LIN {X 0,Y 186.458,Z 664.253,A -85,B 0,C 180,E1 -22354.51,E2 -22354.51} C_VEL
LIN {X 0,Y 188.519,Z 666.422,A -85,B 0,C 180,E1 -22355.462,E2 -22355.462} C_VEL
LIN {X 0,Y 189.961,Z 668.387,A -85,B 0,C 180,E1 -22356.131,E2 -22356.131} C_VEL
LIN {X 0,Y 193.772,Z 674.141,A -85,B 0,C 180,E1 -22357.839,E2 -22357.839} C_VEL
LIN {X 0,Y 198,Z 681.171,A -85,B 0,C 180,E1 -22359.627,E2 -22359.627} C_VEL
LIN {X 0,Y 202.989,Z 690.013,A -85,B 0,C 180,E1 -22361.599,E2 -22361.599} C_VEL
LIN {X 0,Y 209.393,Z 702.579,A -85,B 0,C 180,E1 -22363.96,E2 -22363.96} C_VEL
LIN {X 0,Y 214.813,Z 715.083,A -85,B 0,C 180,E1 -22365.866,E2 -22365.866} C_VEL
LIN {X 0,Y 219.093,Z 726.699,A -85,B 0,C 180,E1 -22367.342,E2 -22367.342} C_VEL
LIN {X 0,Y 219.562,Z 732.346,A -85,B 0,C 180,E1 -22367.681,E2 -22367.681} C_VEL
LIN {X 0,Y 219.234,Z 736.244,A -85,B 0,C 180,E1 -22367.773,E2 -22367.773} C_VEL
LIN {X 0,Y 217.38,Z 743.918,A -85,B 0,C 180,E1 -22367.69,E2 -22367.69} C_VEL
LIN {X 0,Y 213.263,Z 757.174,A -85,B 0,C 180,E1 -22367.338,E2 -22367.338} C_VEL
LIN {X 0,Y 212.359,Z 763.033,A -85,B 0,C 180,E1 -22367.387,E2 -22367.387} C_VEL
LIN {X 0,Y 210.033,Z 802.061,A -85,B 0,C 180,E1 -22368.634,E2 -22368.634} C_VEL
LIN {X 0,Y 208.26,Z 816.506,A -85,B 0,C 180,E1 -22369.407,E2 -22369.407} C_VEL
LIN {X 0,Y 205.986,Z 829.249,A -85,B 0,C 180,E1 -22370.387,E2 -22370.387} C_VEL
LIN {X 0,Y 203.017,Z 842.443,A -85,B 0,C 180,E1 -22371.772,E2 -22371.772} C_VEL
LIN {X 0,Y 199.554,Z 855.196,A -85,B 0,C 180,E1 -22373.536,E2 -22373.536} C_VEL
LIN {X 0,Y 196.163,Z 866.216,A -85,B 0,C 180,E1 -22375.49,E2 -22375.49} C_VEL
LIN {X 0,Y 192.35,Z 877.477,A -85,B 0,C 180,E1 -22378.008,E2 -22378.008} C_VEL
LIN {X 0,Y 188.32,Z 888.046,A -85,B 0,C 180,E1 -22380.977,E2 -22380.977} C_VEL
LIN {X 0,Y 184.98,Z 896.778,A -85,B 0,C 180,E1 -22384.092,E2 -22384.092} C_VEL
LIN {X 0,Y 182.131,Z 904.027,A -85,B 0,C 180,E1 -22387.302,E2 -22387.302} C_VEL
LIN {X 0,Y 179.919,Z 910.061,A -85,B 0,C 180,E1 -22390.608,E2 -22390.608} C_VEL
LIN {X 0,Y 178.213,Z 915.047,A -85,B 0,C 180,E1 -22393.975,E2 -22393.975} C_VEL
LIN {X 0,Y 176.719,Z 920.187,A -85,B 0,C 180,E1 -22398.53,E2 -22398.53} C_VEL
LIN {X 0,Y 176.133,Z 923.805,A -85,B 0,C 180,E1 -22403.125,E2 -22403.125} C_VEL
LIN {X 0,Y 176.096,Z 925.996,A -85,B 0,C 180,E1 -22407.712,E2 -22407.712} C_VEL
LIN {X 0,Y 176.209,Z 926.574,A -85,B 0,C 180,E1 -22410,E2 -22410} C_VEL
LIN {X 0,Y 176.02,Z 926.688,A -85,B 0,C 180,E1 -22414.58,E2 -22414.58} C_VEL
LIN {X 0,Y 176.329,Z 925.467,A -85,B 0,C 180,E1 -22419.174,E2 -22419.174} C_VEL
LIN {X 0,Y 177.401,Z 922.904,A -85,B 0,C 180,E1 -22423.751,E2 -22423.751} C_VEL
LIN {X 0,Y 179.558,Z 918.924,A -85,B 0,C 180,E1 -22428.247,E2 -22428.247} C_VEL
LIN {X 0,Y 182.331,Z 913.868,A -85,B 0,C 180,E1 -22432.32,E2 -22432.32} C_VEL
LIN {X 0,Y 186.083,Z 907.172,A -85,B 0,C 180,E1 -22436.345,E2 -22436.345} C_VEL
LIN {X 0,Y 190.386,Z 899.447,A -85,B 0,C 180,E1 -22439.89,E2 -22439.89} C_VEL
LIN {X 0,Y 194.724,Z 891.411,A -85,B 0,C 180,E1 -22442.778,E2 -22442.778} C_VEL
LIN {X 0,Y 199.516,Z 881.745,A -85,B 0,C 180,E1 -22445.536,E2 -22445.536} C_VEL
LIN {X 0,Y 204.224,Z 871.045,A -85,B 0,C 180,E1 -22447.961,E2 -22447.961} C_VEL
LIN {X 0,Y 208.917,Z 859.221,A -85,B 0,C 180,E1 -22450.043,E2 -22450.043} C_VEL
LIN {X 0,Y 213.409,Z 846.062,A -85,B 0,C 180,E1 -22451.826,E2 -22451.826} C_VEL
LIN {X 0,Y 217.08,Z 833.039,A -85,B 0,C 180,E1 -22453.151,E2 -22453.151} C_VEL
LIN {X 0,Y 220.206,Z 818.846,A -85,B 0,C 180,E1 -22454.199,E2 -22454.199} C_VEL
LIN {X 0,Y 222.422,Z 804.381,A -85,B 0,C 180,E1 -22454.941,E2 -22454.941} C_VEL
LIN {X 0,Y 224.005,Z 785.386,A -85,B 0,C 180,E1 -22455.543,E2 -22455.543} C_VEL
LIN {X 0,Y 226.866,Z 740.906,A -85,B 0,C 180,E1 -22456.815,E2 -22456.815} C_VEL
LIN {X 0,Y 223.203,Z 731.743,A -85,B 0,C 180,E1 -22458.353,E2 -22458.353} C_VEL
LIN {X 0,Y 218.442,Z 721.156,A -85,B 0,C 180,E1 -22460.444,E2 -22460.444} C_VEL
LIN {X 0,Y 212.911,Z 710.324,A -85,B 0,C 180,E1 -22463.05,E2 -22463.05} C_VEL
LIN {X 0,Y 207.489,Z 700.825,A -85,B 0,C 180,E1 -22465.86,E2 -22465.86} C_VEL
LIN {X 0,Y 204.073,Z 695.198,A -85,B 0,C 180,E1 -22467.81,E2 -22467.81} C_VEL
LIN {X 0,Y 201.093,Z 690.54,A -85,B 0,C 180,E1 -22469.652,E2 -22469.652} C_VEL
LIN {X 0,Y 197.75,Z 685.547,A -85,B 0,C 180,E1 -22471.914,E2 -22471.914} C_VEL
LIN {X 0,Y 193.988,Z 680.428,A -85,B 0,C 180,E1 -22474.764,E2 -22474.764} C_VEL
LIN {X 0,Y 193.438,Z 679.67,A -85,B 0,C 180,E1 -22475.22,E2 -22475.22} C_VEL
LIN {X 0,Y 190.753,Z 677.183,A -85,B 0,C 180,E1 -22477.501,E2 -22477.501} C_VEL
LIN {X 0,Y 189.274,Z 674.416,A -85,B 0,C 180,E1 -22479.061,E2 -22479.061} C_VEL
LIN {X 0,Y 186.17,Z 672.169,A -85,B 0,C 180,E1 -22482.423,E2 -22482.423} C_VEL
LIN {X 0,Y 184.562,Z 669.313,A -85,B 0,C 180,E1 -22484.824,E2 -22484.824} C_VEL
LIN {X 0,Y 184.282,Z 668.398,A -85,B 0,C 180,E1 -22485.366,E2 -22485.366} C_VEL
LIN {X 0,Y 180.317,Z 665.407,A -85,B 0,C 180,E1 -22497.767,E2 -22497.767} C_VEL
LIN {X 0,Y 180.526,Z 665.448,A -85,B 0,C 180,E1 -22500.558,E2 -22500.558} C_VEL
LIN {X 0,Y 182.784,Z 667.786,A -85,B 0,C 180,E1 -22507.735,E2 -22507.735} C_VEL
LIN {X 0,Y 184.46,Z 668.55,A -85,B 0,C 180,E1 -22510.486,E2 -22510.486} C_VEL
LIN {X 0,Y 185.451,Z 671.116,A -85,B 0,C 180,E1 -22512.17,E2 -22512.17} C_VEL
LIN {X 0,Y 187.688,Z 673.465,A -85,B 0,C 180,E1 -22514.919,E2 -22514.919} C_VEL
LIN {X 0,Y 189.332,Z 674.523,A -85,B 0,C 180,E1 -22516.581,E2 -22516.581} C_VEL
LIN {X 0,Y 191.05,Z 677.607,A -85,B 0,C 180,E1 -22518.36,E2 -22518.36} C_VEL
LIN {X 0,Y 193.858,Z 680.189,A -85,B 0,C 180,E1 -22520.7,E2 -22520.7} C_VEL
LIN {X 0,Y 196.314,Z 683.711,A -85,B 0,C 180,E1 -22522.635,E2 -22522.635} C_VEL
LIN {X 0,Y 198.092,Z 685.527,A -85,B 0,C 180,E1 -22523.864,E2 -22523.864} C_VEL
LIN {X 0,Y 200.895,Z 689.24,A -85,B 0,C 180,E1 -22525.723,E2 -22525.723} C_VEL
LIN {X 0,Y 205.468,Z 695.423,A -85,B 0,C 180,E1 -22528.447,E2 -22528.447} C_VEL
LIN {X 0,Y 210.739,Z 702.824,A -85,B 0,C 180,E1 -22531.222,E2 -22531.222} C_VEL
LIN {X 0,Y 217.232,Z 712.976,A -85,B 0,C 180,E1 -22534.274,E2 -22534.274} C_VEL
LIN {X 0,Y 223.438,Z 723.698,A -85,B 0,C 180,E1 -22536.899,E2 -22536.899} C_VEL
LIN {X 0,Y 227.451,Z 731.558,A -85,B 0,C 180,E1 -22538.491,E2 -22538.491} C_VEL
LIN {X 0,Y 223.562,Z 789.522,A -85,B 0,C 180,E1 -22540.18,E2 -22540.18} C_VEL
LIN {X 0,Y 221.655,Z 803.905,A -85,B 0,C 180,E1 -22540.886,E2 -22540.886} C_VEL
LIN {X 0,Y 218.999,Z 817.921,A -85,B 0,C 180,E1 -22541.916,E2 -22541.916} C_VEL
LIN {X 0,Y 215.767,Z 830.231,A -85,B 0,C 180,E1 -22543.083,E2 -22543.083} C_VEL
LIN {X 0,Y 211.746,Z 843.508,A -85,B 0,C 180,E1 -22544.81,E2 -22544.81} C_VEL
LIN {X 0,Y 207.507,Z 854.961,A -85,B 0,C 180,E1 -22546.698,E2 -22546.698} C_VEL
LIN {X 0,Y 203.105,Z 865.457,A -85,B 0,C 180,E1 -22548.894,E2 -22548.894} C_VEL
LIN {X 0,Y 198.737,Z 874.93,A -85,B 0,C 180,E1 -22551.396,E2 -22551.396} C_VEL
LIN {X 0,Y 193.842,Z 884.419,A -85,B 0,C 180,E1 -22554.543,E2 -22554.543} C_VEL
LIN {X 0,Y 189.238,Z 892.563,A -85,B 0,C 180,E1 -22558.047,E2 -22558.047} C_VEL
LIN {X 0,Y 185.363,Z 899.091,A -85,B 0,C 180,E1 -22561.71,E2 -22561.71} C_VEL
LIN {X 0,Y 181.765,Z 904.858,A -85,B 0,C 180,E1 -22566.047,E2 -22566.047} C_VEL
LIN {X 0,Y 179.351,Z 908.731,A -85,B 0,C 180,E1 -22570.131,E2 -22570.131} C_VEL
LIN {X 0,Y 177.673,Z 911.216,A -85,B 0,C 180,E1 -22573.926,E2 -22573.926} C_VEL
LIN {X 0,Y 176.494,Z 912.899,A -85,B 0,C 180,E1 -22578.516,E2 -22578.516} C_VEL
LIN {X 0,Y 176.125,Z 913.253,A -85,B 0,C 180,E1 -22583.125,E2 -22583.125} C_VEL
LIN {X 0,Y 176.143,Z 912.827,A -85,B 0,C 180,E1 -22585.948,E2 -22585.948} C_VEL
LIN {X 0,Y 176.326,Z 911.339,A -85,B 0,C 180,E1 -22590,E2 -22590} C_VEL
LIN {X 0,Y 177.015,Z 908.405,A -85,B 0,C 180,E1 -22594.555,E2 -22594.555} C_VEL
LIN {X 0,Y 178.587,Z 904.042,A -85,B 0,C 180,E1 -22599.057,E2 -22599.057} C_VEL
LIN {X 0,Y 180.536,Z 898.946,A -85,B 0,C 180,E1 -22602.919,E2 -22602.919} C_VEL
LIN {X 0,Y 183.049,Z 892.471,A -85,B 0,C 180,E1 -22606.736,E2 -22606.736} C_VEL
LIN {X 0,Y 186.249,Z 884.467,A -85,B 0,C 180,E1 -22610.429,E2 -22610.429} C_VEL
LIN {X 0,Y 189.769,Z 876.064,A -85,B 0,C 180,E1 -22613.461,E2 -22613.461} C_VEL
LIN {X 0,Y 193.576,Z 865.93,A -85,B 0,C 180,E1 -22616.408,E2 -22616.408} C_VEL
LIN {X 0,Y 197.334,Z 854.598,A -85,B 0,C 180,E1 -22619.029,E2 -22619.029} C_VEL
LIN {X 0,Y 200.212,Z 844.74,A -85,B 0,C 180,E1 -22620.889,E2 -22620.889} C_VEL
LIN {X 0,Y 203.414,Z 832.733,A -85,B 0,C 180,E1 -22622.674,E2 -22622.674} C_VEL
LIN {X 0,Y 206.431,Z 819.424,A -85,B 0,C 180,E1 -22624.177,E2 -22624.177} C_VEL
LIN {X 0,Y 208.689,Z 805.589,A -85,B 0,C 180,E1 -22625.368,E2 -22625.368} C_VEL
LIN {X 0,Y 210.399,Z 791.062,A -85,B 0,C 180,E1 -22626.216,E2 -22626.216} C_VEL
LIN {X 0,Y 211.902,Z 767.428,A -85,B 0,C 180,E1 -22627.019,E2 -22627.019} C_VEL
LIN {X 0,Y 214.604,Z 720.39,A -85,B 0,C 180,E1 -22628.444,E2 -22628.444} C_VEL
LIN {X 0,Y 209.401,Z 709.666,A -85,B 0,C 180,E1 -22630.204,E2 -22630.204} C_VEL
LIN {X 0,Y 203.348,Z 698.745,A -85,B 0,C 180,E1 -22632.36,E2 -22632.36} C_VEL
LIN {X 0,Y 197.061,Z 688.675,A -85,B 0,C 180,E1 -22634.769,E2 -22634.769} C_VEL
LIN {X 0,Y 191.638,Z 680.859,A -85,B 0,C 180,E1 -22637.025,E2 -22637.025} C_VEL
LIN {X 0,Y 188.675,Z 676.773,A -85,B 0,C 180,E1 -22638.35,E2 -22638.35} C_VEL
LIN {X 0,Y 186.132,Z 673.147,A -85,B 0,C 180,E1 -22639.561,E2 -22639.561} C_VEL
LIN {X 0,Y 183.199,Z 669.724,A -85,B 0,C 180,E1 -22640.994,E2 -22640.994} C_VEL
LIN {X 0,Y 181.985,Z 667.637,A -85,B 0,C 180,E1 -22641.66,E2 -22641.66} C_VEL
LIN {X 0,Y 179.787,Z 665.649,A -85,B 0,C 180,E1 -22642.793,E2 -22642.793} C_VEL
LIN {X 0,Y 178.655,Z 663.464,A -85,B 0,C 180,E1 -22643.483,E2 -22643.483} C_VEL
LIN {X 0,Y 178.43,Z 662.343,A -85,B 0,C 180,E1 -22643.733,E2 -22643.733} C_VEL
LIN {X 0,Y 178.486,Z 662.376,A -85,B 0,C 180,E1 -22646.546,E2 -22646.546} C_VEL
LIN {X 0,Y 178.447,Z 662.375,A -85,B 0,C 180,E1 -22651.795,E2 -22651.795} C_VEL
LIN {X 0,Y 178.518,Z 662.354,A -85,B 0,C 180,E1 -22654.888,E2 -22654.888} C_VEL
LIN {X 0,Y 178.593,Z 662.347,A -85,B 0,C 180,E1 -22660.814,E2 -22660.814} C_VEL
LIN {X 0,Y 178.647,Z 662.356,A -85,B 0,C 180,E1 -22666.346,E2 -22666.346} C_VEL
LIN {X 0,Y 178.909,Z 662.303,A -85,B 0,C 180,E1 -22670.959,E2 -22670.959} C_VEL
LIN {X 0,Y 179.149,Z 662.292,A -85,B 0,C 180,E1 -22677.751,E2 -22677.751} C_VEL
LIN {X 0,Y 179.369,Z 662.257,A -85,B 0,C 180,E1 -22679.999,E2 -22679.999} C_VEL
LIN {X 0,Y 178.869,Z 662.325,A -85,B 0,C 180,E1 -22684.506,E2 -22684.506} C_VEL
LIN {X 0,Y 178.914,Z 662.322,A -85,B 0,C 180,E1 -22689.04,E2 -22689.04} C_VEL
LIN {X 0,Y 178.66,Z 662.352,A -85,B 0,C 180,E1 -22693.651,E2 -22693.651} C_VEL
LIN {X 0,Y 178.623,Z 662.348,A -85,B 0,C 180,E1 -22699.214,E2 -22699.214} C_VEL
LIN {X 0,Y 178.521,Z 662.367,A -85,B 0,C 180,E1 -22705.114,E2 -22705.114} C_VEL
LIN {X 0,Y 178.524,Z 662.367,A -85,B 0,C 180,E1 -22709.993,E2 -22709.993} C_VEL
LIN {X 0,Y 178.506,Z 662.463,A -85,B 0,C 180,E1 -22710.867,E2 -22710.867} C_VEL
LIN {X 0,Y 179.341,Z 664.986,A -85,B 0,C 180,E1 -22711.445,E2 -22711.445} C_VEL
LIN {X 0,Y 181.355,Z 667.237,A -85,B 0,C 180,E1 -22712.526,E2 -22712.526} C_VEL
LIN {X 0,Y 182.452,Z 668.141,A -85,B 0,C 180,E1 -22713.072,E2 -22713.072} C_VEL
LIN {X 0,Y 184.519,Z 671.443,A -85,B 0,C 180,E1 -22714.168,E2 -22714.168} C_VEL
LIN {X 0,Y 186.456,Z 673.52,A -85,B 0,C 180,E1 -22715.086,E2 -22715.086} C_VEL
LIN {X 0,Y 190.366,Z 679.679,A -85,B 0,C 180,E1 -22716.943,E2 -22716.943} C_VEL
LIN {X 0,Y 195.551,Z 688.346,A -85,B 0,C 180,E1 -22719.219,E2 -22719.219} C_VEL
LIN {X 0,Y 202.299,Z 701.307,A -85,B 0,C 180,E1 -22721.96,E2 -22721.96} C_VEL
LIN {X 0,Y 207.489,Z 712.568,A -85,B 0,C 180,E1 -22723.928,E2 -22723.928} C_VEL
LIN {X 0,Y 212.727,Z 726.005,A -85,B 0,C 180,E1 -22725.851,E2 -22725.851} C_VEL
LIN {X 0,Y 213.798,Z 728.909,A -85,B 0,C 180,E1 -22726.233,E2 -22726.233} C_VEL
LIN {X 0,Y 214.071,Z 733.929,A -85,B 0,C 180,E1 -22726.516,E2 -22726.516} C_VEL
LIN {X 0,Y 212.359,Z 763.033,A -85,B 0,C 180,E1 -22727.387,E2 -22727.387} C_VEL
LIN {X 0,Y 211.505,Z 768.882,A -85,B 0,C 180,E1 -22727.446,E2 -22727.446} C_VEL
LIN {X 0,Y 206.057,Z 787.91,A -85,B 0,C 180,E1 -22727.022,E2 -22727.022} C_VEL
LIN {X 0,Y 205.193,Z 793.759,A -85,B 0,C 180,E1 -22727.081,E2 -22727.081} C_VEL
LIN {X 0,Y 203.858,Z 808.138,A -85,B 0,C 180,E1 -22727.674,E2 -22727.674} C_VEL
LIN {X 0,Y 201.992,Z 820.575,A -85,B 0,C 180,E1 -22728.451,E2 -22728.451} C_VEL
LIN {X 0,Y 199.378,Z 833.862,A -85,B 0,C 180,E1 -22729.63,E2 -22729.63} C_VEL
LIN {X 0,Y 196.088,Z 846.803,A -85,B 0,C 180,E1 -22731.154,E2 -22731.154} C_VEL
LIN {X 0,Y 192.546,Z 858.647,A -85,B 0,C 180,E1 -22732.968,E2 -22732.968} C_VEL
LIN {X 0,Y 188.817,Z 870.156,A -85,B 0,C 180,E1 -22735.25,E2 -22735.25} C_VEL
LIN {X 0,Y 185.62,Z 878.854,A -85,B 0,C 180,E1 -22737.348,E2 -22737.348} C_VEL
LIN {X 0,Y 181.46,Z 889.094,A -85,B 0,C 180,E1 -22740.408,E2 -22740.408} C_VEL
LIN {X 0,Y 178.042,Z 897.603,A -85,B 0,C 180,E1 -22743.635,E2 -22743.635} C_VEL
LIN {X 0,Y 174.615,Z 905.718,A -85,B 0,C 180,E1 -22747.519,E2 -22747.519} C_VEL
LIN {X 0,Y 172.492,Z 911.452,A -85,B 0,C 180,E1 -22750.976,E2 -22750.976} C_VEL
LIN {X 0,Y 170.827,Z 916.103,A -85,B 0,C 180,E1 -22754.489,E2 -22754.489} C_VEL
LIN {X 0,Y 169.453,Z 920.907,A -85,B 0,C 180,E1 -22759.243,E2 -22759.243} C_VEL
LIN {X 0,Y 169.057,Z 923.473,A -85,B 0,C 180,E1 -22762.835,E2 -22762.835} C_VEL
LIN {X 0,Y 168.994,Z 925.69,A -85,B 0,C 180,E1 -22767.616,E2 -22767.616} C_VEL
LIN {X 0,Y 169.112,Z 926.281,A -85,B 0,C 180,E1 -22770,E2 -22770} C_VEL
LIN {X 0,Y 168.932,Z 926.42,A -85,B 0,C 180,E1 -22774.773,E2 -22774.773} C_VEL
LIN {X 0,Y 169.295,Z 925.224,A -85,B 0,C 180,E1 -22779.558,E2 -22779.558} C_VEL
LIN {X 0,Y 170.464,Z 922.687,A -85,B 0,C 180,E1 -22784.322,E2 -22784.322} C_VEL
LIN {X 0,Y 172.771,Z 918.745,A -85,B 0,C 180,E1 -22788.991,E2 -22788.991} C_VEL
LIN {X 0,Y 175.496,Z 914.111,A -85,B 0,C 180,E1 -22792.918,E2 -22792.918} C_VEL
LIN {X 0,Y 179.725,Z 907.059,A -85,B 0,C 180,E1 -22797.353,E2 -22797.353} C_VEL
LIN {X 0,Y 184.214,Z 899.369,A -85,B 0,C 180,E1 -22801,E2 -22801} C_VEL
LIN {X 0,Y 188.784,Z 891.375,A -85,B 0,C 180,E1 -22803.946,E2 -22803.946} C_VEL
LIN {X 0,Y 193.712,Z 881.88,A -85,B 0,C 180,E1 -22806.727,E2 -22806.727} C_VEL
LIN {X 0,Y 198.666,Z 871.113,A -85,B 0,C 180,E1 -22809.223,E2 -22809.223} C_VEL
LIN {X 0,Y 203.548,Z 859.36,A -85,B 0,C 180,E1 -22811.325,E2 -22811.325} C_VEL
LIN {X 0,Y 208.19,Z 846.294,A -85,B 0,C 180,E1 -22813.125,E2 -22813.125} C_VEL
LIN {X 0,Y 211.972,Z 833.429,A -85,B 0,C 180,E1 -22814.459,E2 -22814.459} C_VEL
LIN {X 0,Y 215.043,Z 820.268,A -85,B 0,C 180,E1 -22815.469,E2 -22815.469} C_VEL
LIN {X 0,Y 217.468,Z 805.727,A -85,B 0,C 180,E1 -22816.247,E2 -22816.247} C_VEL
LIN {X 0,Y 218.974,Z 790.136,A -85,B 0,C 180,E1 -22816.771,E2 -22816.771} C_VEL
LIN {X 0,Y 222.095,Z 743.272,A -85,B 0,C 180,E1 -22818.126,E2 -22818.126} C_VEL
LIN {X 0,Y 217.885,Z 732.803,A -85,B 0,C 180,E1 -22820.019,E2 -22820.019} C_VEL
LIN {X 0,Y 213.283,Z 722.763,A -85,B 0,C 180,E1 -22822.198,E2 -22822.198} C_VEL
LIN {X 0,Y 208.354,Z 713.066,A -85,B 0,C 180,E1 -22824.719,E2 -22824.719} C_VEL
LIN {X 0,Y 203.97,Z 705.311,A -85,B 0,C 180,E1 -22827.17,E2 -22827.17} C_VEL
LIN {X 0,Y 200.593,Z 699.584,A -85,B 0,C 180,E1 -22829.25,E2 -22829.25} C_VEL
LIN {X 0,Y 198.46,Z 696.211,A -85,B 0,C 180,E1 -22830.658,E2 -22830.658} C_VEL
LIN {X 0,Y 195.503,Z 691.615,A -85,B 0,C 180,E1 -22832.779,E2 -22832.779} C_VEL
LIN {X 0,Y 191.604,Z 686.244,A -85,B 0,C 180,E1 -22835.917,E2 -22835.917} C_VEL
LIN {X 0,Y 188.948,Z 683.515,A -85,B 0,C 180,E1 -22838.313,E2 -22838.313} C_VEL
LIN {X 0,Y 187.435,Z 681.013,A -85,B 0,C 180,E1 -22839.964,E2 -22839.964} C_VEL
LIN {X 0,Y 184.613,Z 678.641,A -85,B 0,C 180,E1 -22843.269,E2 -22843.269} C_VEL
LIN {X 0,Y 183.101,Z 675.569,A -85,B 0,C 180,E1 -22845.766,E2 -22845.766} C_VEL
LIN {X 0,Y 179.686,Z 673.153,A -85,B 0,C 180,E1 -22854.389,E2 -22854.389} C_VEL
LIN {X 0,Y 179.601,Z 672.339,A -85,B 0,C 180,E1 -22860.001,E2 -22860.001} C_VEL
LIN {X 0,Y 181.924,Z 674.842,A -85,B 0,C 180,E1 -22867.771,E2 -22867.771} C_VEL
LIN {X 0,Y 183.191,Z 675.569,A -85,B 0,C 180,E1 -22869.943,E2 -22869.943} C_VEL
LIN {X 0,Y 184.584,Z 678.556,A -85,B 0,C 180,E1 -22872.263,E2 -22872.263} C_VEL
LIN {X 0,Y 187.337,Z 680.874,A -85,B 0,C 180,E1 -22875.504,E2 -22875.504} C_VEL
LIN {X 0,Y 187.98,Z 681.808,A -85,B 0,C 180,E1 -22876.215,E2 -22876.215} C_VEL
LIN {X 0,Y 190.063,Z 684.904,A -85,B 0,C 180,E1 -22878.337,E2 -22878.337} C_VEL
LIN {X 0,Y 192.078,Z 686.809,A -85,B 0,C 180,E1 -22880.062,E2 -22880.062} C_VEL
LIN {X 0,Y 194.818,Z 690.598,A -85,B 0,C 180,E1 -22882.277,E2 -22882.277} C_VEL
LIN {X 0,Y 196.181,Z 692.185,A -85,B 0,C 180,E1 -22883.265,E2 -22883.265} C_VEL
LIN {X 0,Y 199.998,Z 697.331,A -85,B 0,C 180,E1 -22885.847,E2 -22885.847} C_VEL
LIN {X 0,Y 203.075,Z 701.642,A -85,B 0,C 180,E1 -22887.727,E2 -22887.727} C_VEL
LIN {X 0,Y 208.122,Z 708.931,A -85,B 0,C 180,E1 -22890.504,E2 -22890.504} C_VEL
LIN {X 0,Y 214.273,Z 718.835,A -85,B 0,C 180,E1 -22893.527,E2 -22893.527} C_VEL
LIN {X 0,Y 220.29,Z 729.605,A -85,B 0,C 180,E1 -22896.191,E2 -22896.191} C_VEL
LIN {X 0,Y 222.66,Z 734.201,A -85,B 0,C 180,E1 -22897.178,E2 -22897.178} C_VEL
LIN {X 0,Y 218.857,Z 789.332,A -85,B 0,C 180,E1 -22898.8,E2 -22898.8} C_VEL
LIN {X 0,Y 216.906,Z 803.789,A -85,B 0,C 180,E1 -22899.507,E2 -22899.507} C_VEL
LIN {X 0,Y 214.278,Z 817.335,A -85,B 0,C 180,E1 -22900.491,E2 -22900.491} C_VEL
LIN {X 0,Y 210.729,Z 830.54,A -85,B 0,C 180,E1 -22901.741,E2 -22901.741} C_VEL
LIN {X 0,Y 206.751,Z 843.239,A -85,B 0,C 180,E1 -22903.399,E2 -22903.399} C_VEL
LIN {X 0,Y 202.38,Z 854.789,A -85,B 0,C 180,E1 -22905.315,E2 -22905.315} C_VEL
LIN {X 0,Y 197.755,Z 865.36,A -85,B 0,C 180,E1 -22907.527,E2 -22907.527} C_VEL
LIN {X 0,Y 192.911,Z 875.388,A -85,B 0,C 180,E1 -22910.207,E2 -22910.207} C_VEL
LIN {X 0,Y 188.047,Z 884.44,A -85,B 0,C 180,E1 -22913.275,E2 -22913.275} C_VEL
LIN {X 0,Y 183.178,Z 892.646,A -85,B 0,C 180,E1 -22916.857,E2 -22916.857} C_VEL
LIN {X 0,Y 179.043,Z 899.214,A -85,B 0,C 180,E1 -22920.616,E2 -22920.616} C_VEL
LIN {X 0,Y 175.213,Z 905.016,A -85,B 0,C 180,E1 -22925.092,E2 -22925.092} C_VEL
LIN {X 0,Y 172.472,Z 909.127,A -85,B 0,C 180,E1 -22929.592,E2 -22929.592} C_VEL
LIN {X 0,Y 170.8,Z 911.438,A -85,B 0,C 180,E1 -22933.26,E2 -22933.26} C_VEL
LIN {X 0,Y 169.479,Z 913.152,A -85,B 0,C 180,E1 -22938.034,E2 -22938.034} C_VEL
LIN {X 0,Y 169.045,Z 913.534,A -85,B 0,C 180,E1 -22942.835,E2 -22942.835} C_VEL
LIN {X 0,Y 169.077,Z 912.614,A -85,B 0,C 180,E1 -22947.618,E2 -22947.618} C_VEL
LIN {X 0,Y 169.524,Z 910.383,A -85,B 0,C 180,E1 -22952.376,E2 -22952.376} C_VEL
LIN {X 0,Y 170.681,Z 906.781,A -85,B 0,C 180,E1 -22957.096,E2 -22957.096} C_VEL
LIN {X 0,Y 172.752,Z 901.691,A -85,B 0,C 180,E1 -22961.737,E2 -22961.737} C_VEL
LIN {X 0,Y 174.751,Z 896.764,A -85,B 0,C 180,E1 -22965.153,E2 -22965.153} C_VEL
LIN {X 0,Y 177.612,Z 889.715,A -85,B 0,C 180,E1 -22969.054,E2 -22969.054} C_VEL
LIN {X 0,Y 180.81,Z 882.326,A -85,B 0,C 180,E1 -22972.271,E2 -22972.271} C_VEL
LIN {X 0,Y 184.572,Z 873.445,A -85,B 0,C 180,E1 -22975.364,E2 -22975.364} C_VEL
LIN {X 0,Y 188.689,Z 862.702,A -85,B 0,C 180,E1 -22978.353,E2 -22978.353} C_VEL
LIN {X 0,Y 192.289,Z 851.825,A -85,B 0,C 180,E1 -22980.777,E2 -22980.777} C_VEL
LIN {X 0,Y 195.876,Z 839.885,A -85,B 0,C 180,E1 -22982.867,E2 -22982.867} C_VEL
LIN {X 0,Y 198.795,Z 828.415,A -85,B 0,C 180,E1 -22984.448,E2 -22984.448} C_VEL
LIN {X 0,Y 201.726,Z 814.928,A -85,B 0,C 180,E1 -22985.855,E2 -22985.855} C_VEL
LIN {X 0,Y 203.794,Z 801.653,A -85,B 0,C 180,E1 -22986.89,E2 -22986.89} C_VEL
LIN {X 0,Y 205.301,Z 786.999,A -85,B 0,C 180,E1 -22987.651,E2 -22987.651} C_VEL
LIN {X 0,Y 209.247,Z 722.727,A -85,B 0,C 180,E1 -22989.643,E2 -22989.643} C_VEL
LIN {X 0,Y 203.17,Z 710.55,A -85,B 0,C 180,E1 -22991.831,E2 -22991.831} C_VEL
LIN {X 0,Y 197.493,Z 700.495,A -85,B 0,C 180,E1 -22994.011,E2 -22994.011} C_VEL
LIN {X 0,Y 191.161,Z 690.495,A -85,B 0,C 180,E1 -22996.645,E2 -22996.645} C_VEL
LIN {X 0,Y 185.469,Z 682.376,A -85,B 0,C 180,E1 -22999.253,E2 -22999.253} C_VEL
LIN {X 0,Y 182.417,Z 678.252,A -85,B 0,C 180,E1 -23000.773,E2 -23000.773} C_VEL
LIN {X 0,Y 179.852,Z 674.847,A -85,B 0,C 180,E1 -23002.13,E2 -23002.13} C_VEL
LIN {X 0,Y 179.006,Z 673.631,A -85,B 0,C 180,E1 -23002.603,E2 -23002.603} C_VEL
LIN {X 0,Y 176.473,Z 670.775,A -85,B 0,C 180,E1 -23004.025,E2 -23004.025} C_VEL
LIN {X 0,Y 175.309,Z 668.733,A -85,B 0,C 180,E1 -23004.766,E2 -23004.766} C_VEL
LIN {X 0,Y 172.811,Z 666.643,A -85,B 0,C 180,E1 -23006.262,E2 -23006.262} C_VEL
LIN {X 0,Y 171.611,Z 664.237,A -85,B 0,C 180,E1 -23007.136,E2 -23007.136} C_VEL
LIN {X 0,Y 171.392,Z 663.259,A -85,B 0,C 180,E1 -23007.438,E2 -23007.438} C_VEL
LIN {X 0,Y 171.411,Z 663.24,A -85,B 0,C 180,E1 -23010.526,E2 -23010.526} C_VEL
LIN {X 0,Y 171.443,Z 663.231,A -85,B 0,C 180,E1 -23015.799,E2 -23015.799} C_VEL
LIN {X 0,Y 171.549,Z 663.223,A -85,B 0,C 180,E1 -23020.867,E2 -23020.867} C_VEL
LIN {X 0,Y 171.562,Z 663.239,A -85,B 0,C 180,E1 -23025.771,E2 -23025.771} C_VEL
LIN {X 0,Y 171.846,Z 663.179,A -85,B 0,C 180,E1 -23030.584,E2 -23030.584} C_VEL
LIN {X 0,Y 171.806,Z 663.197,A -85,B 0,C 180,E1 -23035.306,E2 -23035.306} C_VEL
LIN {X 0,Y 172.332,Z 663.134,A -85,B 0,C 180,E1 -23039.999,E2 -23039.999} C_VEL
LIN {X 0,Y 171.817,Z 663.201,A -85,B 0,C 180,E1 -23044.692,E2 -23044.692} C_VEL
LIN {X 0,Y 171.85,Z 663.197,A -85,B 0,C 180,E1 -23049.414,E2 -23049.414} C_VEL
LIN {X 0,Y 171.577,Z 663.229,A -85,B 0,C 180,E1 -23054.227,E2 -23054.227} C_VEL
LIN {X 0,Y 171.542,Z 663.229,A -85,B 0,C 180,E1 -23059.557,E2 -23059.557} C_VEL
LIN {X 0,Y 171.46,Z 663.25,A -85,B 0,C 180,E1 -23065.609,E2 -23065.609} C_VEL
LIN {X 0,Y 171.423,Z 663.247,A -85,B 0,C 180,E1 -23067.135,E2 -23067.135} C_VEL
LIN {X 0,Y 172.311,Z 665.854,A -85,B 0,C 180,E1 -23067.889,E2 -23067.889} C_VEL
LIN {X 0,Y 174.31,Z 668.093,A -85,B 0,C 180,E1 -23069.157,E2 -23069.157} C_VEL
LIN {X 0,Y 175.691,Z 669.113,A -85,B 0,C 180,E1 -23069.952,E2 -23069.952} C_VEL
LIN {X 0,Y 177.375,Z 672.025,A -85,B 0,C 180,E1 -23071.003,E2 -23071.003} C_VEL
LIN {X 0,Y 179.611,Z 674.311,A -85,B 0,C 180,E1 -23072.217,E2 -23072.217} C_VEL
LIN {X 0,Y 182.176,Z 677.936,A -85,B 0,C 180,E1 -23073.597,E2 -23073.597} C_VEL
LIN {X 0,Y 183.397,Z 679.312,A -85,B 0,C 180,E1 -23074.203,E2 -23074.203} C_VEL
LIN {X 0,Y 187.284,Z 685.65,A -85,B 0,C 180,E1 -23076.147,E2 -23076.147} C_VEL
LIN {X 0,Y 192.111,Z 694.04,A -85,B 0,C 180,E1 -23078.378,E2 -23078.378} C_VEL
LIN {X 0,Y 198.464,Z 706.597,A -85,B 0,C 180,E1 -23081.096,E2 -23081.096} C_VEL
LIN {X 0,Y 203.081,Z 716.893,A -85,B 0,C 180,E1 -23082.946,E2 -23082.946} C_VEL
LIN {X 0,Y 208.507,Z 731.352,A -85,B 0,C 180,E1 -23085.058,E2 -23085.058} C_VEL
LIN {X 0,Y 208.748,Z 734.274,A -85,B 0,C 180,E1 -23085.252,E2 -23085.252} C_VEL
LIN {X 0,Y 205.193,Z 793.759,A -85,B 0,C 180,E1 -23087.081,E2 -23087.081} C_VEL
LIN {X 0,Y 204.234,Z 799.591,A -85,B 0,C 180,E1 -23087.161,E2 -23087.161} C_VEL
LIN {X 0,Y 200.991,Z 808.977,A -85,B 0,C 180,E1 -23087.072,E2 -23087.072} C_VEL
LIN {X 0,Y 197.354,Z 818.224,A -85,B 0,C 180,E1 -23087.103,E2 -23087.103} C_VEL
LIN {X 0,Y 196.239,Z 821.966,A -85,B 0,C 180,E1 -23087.275,E2 -23087.275} C_VEL
LIN {X 0,Y 195.847,Z 823.839,A -85,B 0,C 180,E1 -23087.423,E2 -23087.423} C_VEL
LIN {X 0,Y 192.997,Z 836.945,A -85,B 0,C 180,E1 -23088.698,E2 -23088.698} C_VEL
LIN {X 0,Y 189.624,Z 849.203,A -85,B 0,C 180,E1 -23090.257,E2 -23090.257} C_VEL
LIN {X 0,Y 185.627,Z 861.87,A -85,B 0,C 180,E1 -23092.373,E2 -23092.373} C_VEL
LIN {X 0,Y 181.55,Z 873.318,A -85,B 0,C 180,E1 -23094.842,E2 -23094.842} C_VEL
LIN {X 0,Y 177.398,Z 883.684,A -85,B 0,C 180,E1 -23097.667,E2 -23097.667} C_VEL
LIN {X 0,Y 173.406,Z 893.05,A -85,B 0,C 180,E1 -23100.899,E2 -23100.899} C_VEL
LIN {X 0,Y 170.037,Z 900.854,A -85,B 0,C 180,E1 -23104.279,E2 -23104.279} C_VEL
LIN {X 0,Y 167.135,Z 907.323,A -85,B 0,C 180,E1 -23107.762,E2 -23107.762} C_VEL
LIN {X 0,Y 165.099,Z 912.686,A -85,B 0,C 180,E1 -23111.381,E2 -23111.381} C_VEL
LIN {X 0,Y 163.052,Z 918.327,A -85,B 0,C 180,E1 -23116.286,E2 -23116.286} C_VEL
LIN {X 0,Y 162.23,Z 921.486,A -85,B 0,C 180,E1 -23120.021,E2 -23120.021} C_VEL
LIN {X 0,Y 161.867,Z 924.437,A -85,B 0,C 180,E1 -23125.018,E2 -23125.018} C_VEL
LIN {X 0,Y 161.904,Z 925.385,A -85,B 0,C 180,E1 -23127.512,E2 -23127.512} C_VEL
LIN {X 0,Y 162.017,Z 925.989,A -85,B 0,C 180,E1 -23130,E2 -23130} C_VEL
LIN {X 0,Y 161.845,Z 926.153,A -85,B 0,C 180,E1 -23134.982,E2 -23134.982} C_VEL
LIN {X 0,Y 162.248,Z 924.981,A -85,B 0,C 180,E1 -23139.978,E2 -23139.978} C_VEL
LIN {X 0,Y 163.544,Z 922.47,A -85,B 0,C 180,E1 -23144.942,E2 -23144.942} C_VEL
LIN {X 0,Y 166.023,Z 918.562,A -85,B 0,C 180,E1 -23149.795,E2 -23149.795} C_VEL
LIN {X 0,Y 168.689,Z 914.312,A -85,B 0,C 180,E1 -23153.571,E2 -23153.571} C_VEL
LIN {X 0,Y 172.777,Z 907.919,A -85,B 0,C 180,E1 -23157.89,E2 -23157.89} C_VEL
LIN {X 0,Y 177.429,Z 900.516,A -85,B 0,C 180,E1 -23161.657,E2 -23161.657} C_VEL
LIN {X 0,Y 182.088,Z 892.781,A -85,B 0,C 180,E1 -23164.701,E2 -23164.701} C_VEL
LIN {X 0,Y 187.113,Z 883.716,A -85,B 0,C 180,E1 -23167.534,E2 -23167.534} C_VEL
LIN {X 0,Y 192.251,Z 873.309,A -85,B 0,C 180,E1 -23170.112,E2 -23170.112} C_VEL
LIN {X 0,Y 197.227,Z 862.081,A -85,B 0,C 180,E1 -23172.267,E2 -23172.267} C_VEL
LIN {X 0,Y 202.05,Z 849.687,A -85,B 0,C 180,E1 -23174.081,E2 -23174.081} C_VEL
LIN {X 0,Y 205.9,Z 837.763,A -85,B 0,C 180,E1 -23175.441,E2 -23175.441} C_VEL
LIN {X 0,Y 209.296,Z 824.734,A -85,B 0,C 180,E1 -23176.565,E2 -23176.565} C_VEL
LIN {X 0,Y 212.037,Z 810.794,A -85,B 0,C 180,E1 -23177.423,E2 -23177.423} C_VEL
LIN {X 0,Y 213.921,Z 795.924,A -85,B 0,C 180,E1 -23178.021,E2 -23178.021} C_VEL
LIN {X 0,Y 217.455,Z 745.627,A -85,B 0,C 180,E1 -23179.492,E2 -23179.492} C_VEL
LIN {X 0,Y 212.308,Z 732.921,A -85,B 0,C 180,E1 -23181.987,E2 -23181.987} C_VEL
LIN {X 0,Y 206.473,Z 720.634,A -85,B 0,C 180,E1 -23185.047,E2 -23185.047} C_VEL
LIN {X 0,Y 201.707,Z 711.815,A -85,B 0,C 180,E1 -23187.813,E2 -23187.813} C_VEL
LIN {X 0,Y 197.118,Z 703.631,A -85,B 0,C 180,E1 -23190.837,E2 -23190.837} C_VEL
LIN {X 0,Y 192.893,Z 697.094,A -85,B 0,C 180,E1 -23193.99,E2 -23193.99} C_VEL
LIN {X 0,Y 189.892,Z 692.872,A -85,B 0,C 180,E1 -23196.551,E2 -23196.551} C_VEL
LIN {X 0,Y 187.103,Z 689.718,A -85,B 0,C 180,E1 -23199.228,E2 -23199.228} C_VEL
LIN {X 0,Y 186.052,Z 687.855,A -85,B 0,C 180,E1 -23200.446,E2 -23200.446} C_VEL
LIN {X 0,Y 183.315,Z 685.404,A -85,B 0,C 180,E1 -23203.805,E2 -23203.805} C_VEL
LIN {X 0,Y 181.721,Z 682.292,A -85,B 0,C 180,E1 -23206.583,E2 -23206.583} C_VEL
LIN {X 0,Y 178.668,Z 680.019,A -85,B 0,C 180,E1 -23215.488,E2 -23215.488} C_VEL
LIN {X 0,Y 178.73,Z 679.425,A -85,B 0,C 180,E1 -23220.001,E2 -23220.001} C_VEL
LIN {X 0,Y 181.065,Z 681.902,A -85,B 0,C 180,E1 -23227.809,E2 -23227.809} C_VEL
LIN {X 0,Y 181.929,Z 682.392,A -85,B 0,C 180,E1 -23229.339,E2 -23229.339} C_VEL
LIN {X 0,Y 183.491,Z 685.602,A -85,B 0,C 180,E1 -23232.021,E2 -23232.021} C_VEL
LIN {X 0,Y 186.274,Z 688.153,A -85,B 0,C 180,E1 -23235.385,E2 -23235.385} C_VEL
LIN {X 0,Y 188.366,Z 691.434,A -85,B 0,C 180,E1 -23237.647,E2 -23237.647} C_VEL
LIN {X 0,Y 190.323,Z 693.42,A -85,B 0,C 180,E1 -23239.412,E2 -23239.412} C_VEL
LIN {X 0,Y 193.129,Z 697.27,A -85,B 0,C 180,E1 -23241.761,E2 -23241.761} C_VEL
LIN {X 0,Y 194.387,Z 698.953,A -85,B 0,C 180,E1 -23242.723,E2 -23242.723} C_VEL
LIN {X 0,Y 197.734,Z 703.524,A -85,B 0,C 180,E1 -23245.079,E2 -23245.079} C_VEL
LIN {X 0,Y 201.492,Z 708.94,A -85,B 0,C 180,E1 -23247.457,E2 -23247.457} C_VEL
LIN {X 0,Y 206.866,Z 717.131,A -85,B 0,C 180,E1 -23250.479,E2 -23250.479} C_VEL
LIN {X 0,Y 213.129,Z 727.841,A -85,B 0,C 180,E1 -23253.609,E2 -23253.609} C_VEL
LIN {X 0,Y 217.979,Z 737.091,A -85,B 0,C 180,E1 -23255.815,E2 -23255.815} C_VEL
LIN {X 0,Y 214.218,Z 789.814,A -85,B 0,C 180,E1 -23257.392,E2 -23257.392} C_VEL
LIN {X 0,Y 212.139,Z 804.45,A -85,B 0,C 180,E1 -23258.111,E2 -23258.111} C_VEL
LIN {X 0,Y 209.426,Z 817.896,A -85,B 0,C 180,E1 -23259.101,E2 -23259.101} C_VEL
LIN {X 0,Y 205.752,Z 831.102,A -85,B 0,C 180,E1 -23260.365,E2 -23260.365} C_VEL
LIN {X 0,Y 201.89,Z 842.976,A -85,B 0,C 180,E1 -23261.92,E2 -23261.92} C_VEL
LIN {X 0,Y 197.353,Z 854.621,A -85,B 0,C 180,E1 -23263.852,E2 -23263.852} C_VEL
LIN {X 0,Y 192.526,Z 865.266,A -85,B 0,C 180,E1 -23266.086,E2 -23266.086} C_VEL
LIN {X 0,Y 187.608,Z 874.981,A -85,B 0,C 180,E1 -23268.681,E2 -23268.681} C_VEL
LIN {X 0,Y 182.321,Z 884.458,A -85,B 0,C 180,E1 -23271.92,E2 -23271.92} C_VEL
LIN {X 0,Y 177.199,Z 892.729,A -85,B 0,C 180,E1 -23275.586,E2 -23275.586} C_VEL
LIN {X 0,Y 172.799,Z 899.337,A -85,B 0,C 180,E1 -23279.443,E2 -23279.443} C_VEL
LIN {X 0,Y 168.722,Z 905.173,A -85,B 0,C 180,E1 -23284.064,E2 -23284.064} C_VEL
LIN {X 0,Y 165.559,Z 909.559,A -85,B 0,C 180,E1 -23289.055,E2 -23289.055} C_VEL
LIN {X 0,Y 163.939,Z 911.66,A -85,B 0,C 180,E1 -23292.537,E2 -23292.537} C_VEL
LIN {X 0,Y 162.487,Z 913.404,A -85,B 0,C 180,E1 -23297.511,E2 -23297.511} C_VEL
LIN {X 0,Y 161.958,Z 913.817,A -85,B 0,C 180,E1 -23302.52,E2 -23302.52} C_VEL
LIN {X 0,Y 161.968,Z 913.263,A -85,B 0,C 180,E1 -23306.393,E2 -23306.393} C_VEL
LIN {X 0,Y 162.143,Z 911.99,A -85,B 0,C 180,E1 -23310,E2 -23310} C_VEL
LIN {X 0,Y 162.904,Z 909.118,A -85,B 0,C 180,E1 -23314.95,E2 -23314.95} C_VEL
LIN {X 0,Y 164.625,Z 904.82,A -85,B 0,C 180,E1 -23319.833,E2 -23319.833} C_VEL
LIN {X 0,Y 166.454,Z 900.579,A -85,B 0,C 180,E1 -23323.42,E2 -23323.42} C_VEL
LIN {X 0,Y 168.76,Z 895.381,A -85,B 0,C 180,E1 -23326.949,E2 -23326.949} C_VEL
LIN {X 0,Y 171.941,Z 887.916,A -85,B 0,C 180,E1 -23330.956,E2 -23330.956} C_VEL
LIN {X 0,Y 175.571,Z 880.114,A -85,B 0,C 180,E1 -23334.224,E2 -23334.224} C_VEL
LIN {X 0,Y 179.595,Z 870.711,A -85,B 0,C 180,E1 -23337.375,E2 -23337.375} C_VEL
LIN {X 0,Y 183.528,Z 860.318,A -85,B 0,C 180,E1 -23340.173,E2 -23340.173} C_VEL
LIN {X 0,Y 186.967,Z 850.128,A -85,B 0,C 180,E1 -23342.388,E2 -23342.388} C_VEL
LIN {X 0,Y 190.858,Z 837.655,A -85,B 0,C 180,E1 -23344.483,E2 -23344.483} C_VEL
LIN {X 0,Y 193.969,Z 825.599,A -85,B 0,C 180,E1 -23346.071,E2 -23346.071} C_VEL
LIN {X 0,Y 196.716,Z 812.333,A -85,B 0,C 180,E1 -23347.399,E2 -23347.399} C_VEL
LIN {X 0,Y 198.883,Z 797.864,A -85,B 0,C 180,E1 -23348.442,E2 -23348.442} C_VEL
LIN {X 0,Y 200.251,Z 783.558,A -85,B 0,C 180,E1 -23349.097,E2 -23349.097} C_VEL
LIN {X 0,Y 203.867,Z 725.065,A -85,B 0,C 180,E1 -23350.937,E2 -23350.937} C_VEL
LIN {X 0,Y 197.554,Z 712.411,A -85,B 0,C 180,E1 -23353.373,E2 -23353.373} C_VEL
LIN {X 0,Y 190.354,Z 699.969,A -85,B 0,C 180,E1 -23356.391,E2 -23356.391} C_VEL
LIN {X 0,Y 184.54,Z 691.268,A -85,B 0,C 180,E1 -23359.072,E2 -23359.072} C_VEL
LIN {X 0,Y 179.637,Z 684.254,A -85,B 0,C 180,E1 -23361.589,E2 -23361.589} C_VEL
LIN {X 0,Y 176.839,Z 680.438,A -85,B 0,C 180,E1 -23363.149,E2 -23363.149} C_VEL
LIN {X 0,Y 173.486,Z 676.223,A -85,B 0,C 180,E1 -23365.15,E2 -23365.15} C_VEL
LIN {X 0,Y 172.793,Z 675.032,A -85,B 0,C 180,E1 -23365.612,E2 -23365.612} C_VEL
LIN {X 0,Y 170.172,Z 672.475,A -85,B 0,C 180,E1 -23367.294,E2 -23367.294} C_VEL
LIN {X 0,Y 168.721,Z 669.822,A -85,B 0,C 180,E1 -23368.394,E2 -23368.394} C_VEL
LIN {X 0,Y 166,Z 667.838,A -85,B 0,C 180,E1 -23370.341,E2 -23370.341} C_VEL
LIN {X 0,Y 164.611,Z 665.406,A -85,B 0,C 180,E1 -23371.554,E2 -23371.554} C_VEL
LIN {X 0,Y 164.312,Z 664.136,A -85,B 0,C 180,E1 -23371.933,E2 -23371.933} C_VEL
LIN {X 0,Y 164.397,Z 664.113,A -85,B 0,C 180,E1 -23374.69,E2 -23374.69} C_VEL
LIN {X 0,Y 164.442,Z 664.118,A -85,B 0,C 180,E1 -23380.094,E2 -23380.094} C_VEL
LIN {X 0,Y 164.49,Z 664.114,A -85,B 0,C 180,E1 -23385.145,E2 -23385.145} C_VEL
LIN {X 0,Y 164.767,Z 664.058,A -85,B 0,C 180,E1 -23390.176,E2 -23390.176} C_VEL
LIN {X 0,Y 164.826,Z 664.076,A -85,B 0,C 180,E1 -23392.65,E2 -23392.65} C_VEL
LIN {X 0,Y 165.044,Z 664.047,A -85,B 0,C 180,E1 -23397.559,E2 -23397.559} C_VEL
LIN {X 0,Y 165.295,Z 664.01,A -85,B 0,C 180,E1 -23399.999,E2 -23399.999} C_VEL
LIN {X 0,Y 164.765,Z 664.078,A -85,B 0,C 180,E1 -23404.893,E2 -23404.893} C_VEL
LIN {X 0,Y 164.833,Z 664.072,A -85,B 0,C 180,E1 -23407.348,E2 -23407.348} C_VEL
LIN {X 0,Y 164.705,Z 664.081,A -85,B 0,C 180,E1 -23411.061,E2 -23411.061} C_VEL
LIN {X 0,Y 164.485,Z 664.118,A -85,B 0,C 180,E1 -23417.402,E2 -23417.402} C_VEL
LIN {X 0,Y 164.39,Z 664.129,A -85,B 0,C 180,E1 -23421.967,E2 -23421.967} C_VEL
LIN {X 0,Y 164.365,Z 664.129,A -85,B 0,C 180,E1 -23422.632,E2 -23422.632} C_VEL
LIN {X 0,Y 165.137,Z 666.565,A -85,B 0,C 180,E1 -23423.431,E2 -23423.431} C_VEL
LIN {X 0,Y 167.292,Z 669.007,A -85,B 0,C 180,E1 -23425.122,E2 -23425.122} C_VEL
LIN {X 0,Y 168.909,Z 670.107,A -85,B 0,C 180,E1 -23426.242,E2 -23426.242} C_VEL
LIN {X 0,Y 170.733,Z 673.194,A -85,B 0,C 180,E1 -23427.586,E2 -23427.586} C_VEL
LIN {X 0,Y 173.093,Z 675.438,A -85,B 0,C 180,E1 -23429.075,E2 -23429.075} C_VEL
LIN {X 0,Y 175.664,Z 679.087,A -85,B 0,C 180,E1 -23430.673,E2 -23430.673} C_VEL
LIN {X 0,Y 177.069,Z 680.769,A -85,B 0,C 180,E1 -23431.478,E2 -23431.478} C_VEL
LIN {X 0,Y 181.019,Z 686.131,A -85,B 0,C 180,E1 -23433.636,E2 -23433.636} C_VEL
LIN {X 0,Y 185.869,Z 694.354,A -85,B 0,C 180,E1 -23436.13,E2 -23436.13} C_VEL
LIN {X 0,Y 192.027,Z 706.178,A -85,B 0,C 180,E1 -23439.024,E2 -23439.024} C_VEL
LIN {X 0,Y 197.665,Z 718.533,A -85,B 0,C 180,E1 -23441.468,E2 -23441.468} C_VEL
LIN {X 0,Y 202.937,Z 732.603,A -85,B 0,C 180,E1 -23443.666,E2 -23443.666} C_VEL
LIN {X 0,Y 203.503,Z 734.261,A -85,B 0,C 180,E1 -23443.898,E2 -23443.898} C_VEL
LIN {X 0,Y 199.309,Z 800.872,A -85,B 0,C 180,E1 -23446.035,E2 -23446.035} C_VEL
LIN {X 0,Y 197.55,Z 814.767,A -85,B 0,C 180,E1 -23446.777,E2 -23446.777} C_VEL
LIN {X 0,Y 195.847,Z 823.839,A -85,B 0,C 180,E1 -23447.423,E2 -23447.423} C_VEL
LIN {X 0,Y 194.206,Z 829.397,A -85,B 0,C 180,E1 -23447.782,E2 -23447.782} C_VEL
LIN {X 0,Y 189.898,Z 838.253,A -85,B 0,C 180,E1 -23448.157,E2 -23448.157} C_VEL
LIN {X 0,Y 185.256,Z 846.821,A -85,B 0,C 180,E1 -23448.712,E2 -23448.712} C_VEL
LIN {X 0,Y 183.115,Z 851.91,A -85,B 0,C 180,E1 -23449.362,E2 -23449.362} C_VEL
LIN {X 0,Y 178.94,Z 864.206,A -85,B 0,C 180,E1 -23451.589,E2 -23451.589} C_VEL
LIN {X 0,Y 174.483,Z 875.705,A -85,B 0,C 180,E1 -23454.264,E2 -23454.264} C_VEL
LIN {X 0,Y 169.913,Z 886.438,A -85,B 0,C 180,E1 -23457.472,E2 -23457.472} C_VEL
LIN {X 0,Y 165.904,Z 895.295,A -85,B 0,C 180,E1 -23460.846,E2 -23460.846} C_VEL
LIN {X 0,Y 162.024,Z 903.792,A -85,B 0,C 180,E1 -23464.981,E2 -23464.981} C_VEL
LIN {X 0,Y 159.678,Z 908.924,A -85,B 0,C 180,E1 -23468.127,E2 -23468.127} C_VEL
LIN {X 0,Y 157.099,Z 915.324,A -85,B 0,C 180,E1 -23473.095,E2 -23473.095} C_VEL
LIN {X 0,Y 155.434,Z 920.188,A -85,B 0,C 180,E1 -23478.26,E2 -23478.26} C_VEL
LIN {X 0,Y 154.914,Z 922.808,A -85,B 0,C 180,E1 -23482.177,E2 -23482.177} C_VEL
LIN {X 0,Y 154.814,Z 925.08,A -85,B 0,C 180,E1 -23487.398,E2 -23487.398} C_VEL
LIN {X 0,Y 154.924,Z 925.697,A -85,B 0,C 180,E1 -23490,E2 -23490} C_VEL
LIN {X 0,Y 154.744,Z 925.885,A -85,B 0,C 180,E1 -23495.211,E2 -23495.211} C_VEL
LIN {X 0,Y 155.222,Z 924.738,A -85,B 0,C 180,E1 -23500.434,E2 -23500.434} C_VEL
LIN {X 0,Y 156.645,Z 922.252,A -85,B 0,C 180,E1 -23505.616,E2 -23505.616} C_VEL
LIN {X 0,Y 159.319,Z 918.375,A -85,B 0,C 180,E1 -23510.665,E2 -23510.665} C_VEL
LIN {X 0,Y 162.987,Z 912.952,A -85,B 0,C 180,E1 -23515.543,E2 -23515.543} C_VEL
LIN {X 0,Y 166.503,Z 907.79,A -85,B 0,C 180,E1 -23519.039,E2 -23519.039} C_VEL
LIN {X 0,Y 171.378,Z 900.426,A -85,B 0,C 180,E1 -23522.913,E2 -23522.913} C_VEL
LIN {X 0,Y 177.175,Z 891.305,A -85,B 0,C 180,E1 -23526.513,E2 -23526.513} C_VEL
LIN {X 0,Y 182.749,Z 881.471,A -85,B 0,C 180,E1 -23529.511,E2 -23529.511} C_VEL
LIN {X 0,Y 188.383,Z 870.188,A -85,B 0,C 180,E1 -23532.185,E2 -23532.185} C_VEL
LIN {X 0,Y 193.669,Z 858.359,A -85,B 0,C 180,E1 -23534.311,E2 -23534.311} C_VEL
LIN {X 0,Y 198.097,Z 846.771,A -85,B 0,C 180,E1 -23535.924,E2 -23535.924} C_VEL
LIN {X 0,Y 202.418,Z 833.178,A -85,B 0,C 180,E1 -23537.361,E2 -23537.361} C_VEL
LIN {X 0,Y 205.679,Z 820.121,A -85,B 0,C 180,E1 -23538.371,E2 -23538.371} C_VEL
LIN {X 0,Y 208.314,Z 805.418,A -85,B 0,C 180,E1 -23539.164,E2 -23539.164} C_VEL
LIN {X 0,Y 209.937,Z 789.658,A -85,B 0,C 180,E1 -23539.701,E2 -23539.701} C_VEL
LIN {X 0,Y 212.946,Z 748.208,A -85,B 0,C 180,E1 -23540.903,E2 -23540.903} C_VEL
LIN {X 0,Y 208.138,Z 736.213,A -85,B 0,C 180,E1 -23543.404,E2 -23543.404} C_VEL
LIN {X 0,Y 203.093,Z 725.341,A -85,B 0,C 180,E1 -23546.24,E2 -23546.24} C_VEL
LIN {X 0,Y 198.756,Z 716.989,A -85,B 0,C 180,E1 -23548.934,E2 -23548.934} C_VEL
LIN {X 0,Y 194.612,Z 709.372,A -85,B 0,C 180,E1 -23551.841,E2 -23551.841} C_VEL
LIN {X 0,Y 190.626,Z 702.957,A -85,B 0,C 180,E1 -23555.014,E2 -23555.014} C_VEL
LIN {X 0,Y 188.144,Z 699.431,A -85,B 0,C 180,E1 -23557.25,E2 -23557.25} C_VEL
LIN {X 0,Y 185.398,Z 696.07,A -85,B 0,C 180,E1 -23560.052,E2 -23560.052} C_VEL
LIN {X 0,Y 184.528,Z 694.566,A -85,B 0,C 180,E1 -23561.112,E2 -23561.112} C_VEL
LIN {X 0,Y 181.865,Z 691.875,A -85,B 0,C 180,E1 -23564.622,E2 -23564.622} C_VEL
LIN {X 0,Y 180.555,Z 689.236,A -85,B 0,C 180,E1 -23567.067,E2 -23567.067} C_VEL
LIN {X 0,Y 177.723,Z 686.84,A -85,B 0,C 180,E1 -23576.6,E2 -23576.6} C_VEL
LIN {X 0,Y 177.858,Z 686.513,A -85,B 0,C 180,E1 -23580.001,E2 -23580.001} C_VEL
LIN {X 0,Y 180.206,Z 688.95,A -85,B 0,C 180,E1 -23587.846,E2 -23587.846} C_VEL
LIN {X 0,Y 180.79,Z 689.486,A -85,B 0,C 180,E1 -23588.946,E2 -23588.946} C_VEL
LIN {X 0,Y 182.52,Z 692.769,A -85,B 0,C 180,E1 -23591.945,E2 -23591.945} C_VEL
LIN {X 0,Y 184.813,Z 694.93,A -85,B 0,C 180,E1 -23594.804,E2 -23594.804} C_VEL
LIN {X 0,Y 186.939,Z 698.229,A -85,B 0,C 180,E1 -23597.187,E2 -23597.187} C_VEL
LIN {X 0,Y 188.646,Z 700.086,A -85,B 0,C 180,E1 -23598.797,E2 -23598.797} C_VEL
LIN {X 0,Y 191.437,Z 703.923,A -85,B 0,C 180,E1 -23601.221,E2 -23601.221} C_VEL
LIN {X 0,Y 195.598,Z 709.814,A -85,B 0,C 180,E1 -23604.356,E2 -23604.356} C_VEL
LIN {X 0,Y 200.435,Z 717.116,A -85,B 0,C 180,E1 -23607.508,E2 -23607.508} C_VEL
LIN {X 0,Y 204.561,Z 723.801,A -85,B 0,C 180,E1 -23609.898,E2 -23609.898} C_VEL
LIN {X 0,Y 209.854,Z 733.102,A -85,B 0,C 180,E1 -23612.667,E2 -23612.667} C_VEL
LIN {X 0,Y 213.485,Z 740.257,A -85,B 0,C 180,E1 -23614.43,E2 -23614.43} C_VEL
LIN {X 0,Y 209.733,Z 790.05,A -85,B 0,C 180,E1 -23615.908,E2 -23615.908} C_VEL
LIN {X 0,Y 207.659,Z 804.345,A -85,B 0,C 180,E1 -23616.608,E2 -23616.608} C_VEL
LIN {X 0,Y 204.971,Z 817.318,A -85,B 0,C 180,E1 -23617.543,E2 -23617.543} C_VEL
LIN {X 0,Y 201.333,Z 830.27,A -85,B 0,C 180,E1 -23618.763,E2 -23618.763} C_VEL
LIN {X 0,Y 197.074,Z 842.964,A -85,B 0,C 180,E1 -23620.404,E2 -23620.404} C_VEL
LIN {X 0,Y 192.465,Z 854.455,A -85,B 0,C 180,E1 -23622.316,E2 -23622.316} C_VEL
LIN {X 0,Y 187.423,Z 865.174,A -85,B 0,C 180,E1 -23624.565,E2 -23624.565} C_VEL
LIN {X 0,Y 181.938,Z 875.567,A -85,B 0,C 180,E1 -23627.377,E2 -23627.377} C_VEL
LIN {X 0,Y 176.711,Z 884.478,A -85,B 0,C 180,E1 -23630.481,E2 -23630.481} C_VEL
LIN {X 0,Y 171.3,Z 892.806,A -85,B 0,C 180,E1 -23634.223,E2 -23634.223} C_VEL
LIN {X 0,Y 166.641,Z 899.46,A -85,B 0,C 180,E1 -23638.185,E2 -23638.185} C_VEL
LIN {X 0,Y 162.268,Z 905.332,A -85,B 0,C 180,E1 -23642.95,E2 -23642.95} C_VEL
LIN {X 0,Y 159.686,Z 908.715,A -85,B 0,C 180,E1 -23646.665,E2 -23646.665} C_VEL
LIN {X 0,Y 157.097,Z 911.883,A -85,B 0,C 180,E1 -23651.751,E2 -23651.751} C_VEL
LIN {X 0,Y 155.497,Z 913.657,A -85,B 0,C 180,E1 -23656.939,E2 -23656.939} C_VEL
LIN {X 0,Y 154.895,Z 914.099,A -85,B 0,C 180,E1 -23662.177,E2 -23662.177} C_VEL
LIN {X 0,Y 154.887,Z 913.236,A -85,B 0,C 180,E1 -23667.4,E2 -23667.4} C_VEL
LIN {X 0,Y 155.378,Z 911.064,A -85,B 0,C 180,E1 -23672.593,E2 -23672.593} C_VEL
LIN {X 0,Y 156.644,Z 907.525,A -85,B 0,C 180,E1 -23677.736,E2 -23677.736} C_VEL
LIN {X 0,Y 158.922,Z 902.503,A -85,B 0,C 180,E1 -23682.775,E2 -23682.775} C_VEL
LIN {X 0,Y 161.046,Z 897.826,A -85,B 0,C 180,E1 -23686.349,E2 -23686.349} C_VEL
LIN {X 0,Y 164.323,Z 890.678,A -85,B 0,C 180,E1 -23690.662,E2 -23690.662} C_VEL
LIN {X 0,Y 167.801,Z 883.38,A -85,B 0,C 180,E1 -23694.102,E2 -23694.102} C_VEL
LIN {X 0,Y 171.918,Z 874.599,A -85,B 0,C 180,E1 -23697.381,E2 -23697.381} C_VEL
LIN {X 0,Y 176.386,Z 863.977,A -85,B 0,C 180,E1 -23700.532,E2 -23700.532} C_VEL
LIN {X 0,Y 180.325,Z 853.245,A -85,B 0,C 180,E1 -23703.068,E2 -23703.068} C_VEL
LIN {X 0,Y 183.707,Z 842.914,A -85,B 0,C 180,E1 -23705.019,E2 -23705.019} C_VEL
LIN {X 0,Y 187.329,Z 830.279,A -85,B 0,C 180,E1 -23706.89,E2 -23706.89} C_VEL
LIN {X 0,Y 190.492,Z 817.173,A -85,B 0,C 180,E1 -23708.337,E2 -23708.337} C_VEL
LIN {X 0,Y 192.825,Z 803.773,A -85,B 0,C 180,E1 -23709.461,E2 -23709.461} C_VEL
LIN {X 0,Y 194.604,Z 789.021,A -85,B 0,C 180,E1 -23710.292,E2 -23710.292} C_VEL
LIN {X 0,Y 198.704,Z 727.696,A -85,B 0,C 180,E1 -23712.254,E2 -23712.254} C_VEL
LIN {X 0,Y 192.231,Z 714.654,A -85,B 0,C 180,E1 -23714.937,E2 -23714.937} C_VEL
LIN {X 0,Y 186.253,Z 704.403,A -85,B 0,C 180,E1 -23717.616,E2 -23717.616} C_VEL
LIN {X 0,Y 180.934,Z 696.195,A -85,B 0,C 180,E1 -23720.236,E2 -23720.236} C_VEL
LIN {X 0,Y 176.17,Z 689.416,A -85,B 0,C 180,E1 -23722.831,E2 -23722.831} C_VEL
LIN {X 0,Y 173.122,Z 685.241,A -85,B 0,C 180,E1 -23724.654,E2 -23724.654} C_VEL
LIN {X 0,Y 169.886,Z 680.931,A -85,B 0,C 180,E1 -23726.762,E2 -23726.762} C_VEL
LIN {X 0,Y 167.346,Z 677.886,A -85,B 0,C 180,E1 -23728.547,E2 -23728.547} C_VEL
LIN {X 0,Y 166.392,Z 676.276,A -85,B 0,C 180,E1 -23729.301,E2 -23729.301} C_VEL
LIN {X 0,Y 163.694,Z 673.881,A -85,B 0,C 180,E1 -23731.38,E2 -23731.38} C_VEL
LIN {X 0,Y 162.07,Z 670.864,A -85,B 0,C 180,E1 -23732.913,E2 -23732.913} C_VEL
LIN {X 0,Y 159.047,Z 668.843,A -85,B 0,C 180,E1 -23735.7,E2 -23735.7} C_VEL
LIN {X 0,Y 157.74,Z 666.639,A -85,B 0,C 180,E1 -23737.227,E2 -23737.227} C_VEL
LIN {X 0,Y 157.327,Z 665.001,A -85,B 0,C 180,E1 -23737.943,E2 -23737.943} C_VEL
LIN {X 0,Y 157.379,Z 664.98,A -85,B 0,C 180,E1 -23741.783,E2 -23741.783} C_VEL
LIN {X 0,Y 157.511,Z 664.98,A -85,B 0,C 180,E1 -23747.108,E2 -23747.108} C_VEL
LIN {X 0,Y 157.689,Z 664.938,A -85,B 0,C 180,E1 -23749.73,E2 -23749.73} C_VEL
LIN {X 0,Y 157.764,Z 664.951,A -85,B 0,C 180,E1 -23752.319,E2 -23752.319} C_VEL
LIN {X 0,Y 158.257,Z 664.886,A -85,B 0,C 180,E1 -23759.999,E2 -23759.999} C_VEL
LIN {X 0,Y 157.77,Z 664.954,A -85,B 0,C 180,E1 -23767.679,E2 -23767.679} C_VEL
LIN {X 0,Y 157.639,Z 664.961,A -85,B 0,C 180,E1 -23771.237,E2 -23771.237} C_VEL
LIN {X 0,Y 157.447,Z 665.161,A -85,B 0,C 180,E1 -23776.782,E2 -23776.782} C_VEL
LIN {X 0,Y 158.227,Z 667.499,A -85,B 0,C 180,E1 -23777.863,E2 -23777.863} C_VEL
LIN {X 0,Y 159.972,Z 669.588,A -85,B 0,C 180,E1 -23779.71,E2 -23779.71} C_VEL
LIN {X 0,Y 162.194,Z 671.026,A -85,B 0,C 180,E1 -23781.694,E2 -23781.694} C_VEL
LIN {X 0,Y 163.815,Z 674.004,A -85,B 0,C 180,E1 -23783.213,E2 -23783.213} C_VEL
LIN {X 0,Y 166.654,Z 676.647,A -85,B 0,C 180,E1 -23785.397,E2 -23785.397} C_VEL
LIN {X 0,Y 168.911,Z 680,A -85,B 0,C 180,E1 -23787.085,E2 -23787.085} C_VEL
LIN {X 0,Y 170.775,Z 681.951,A -85,B 0,C 180,E1 -23788.319,E2 -23788.319} C_VEL
LIN {X 0,Y 173.495,Z 685.599,A -85,B 0,C 180,E1 -23790.06,E2 -23790.06} C_VEL
LIN {X 0,Y 178.148,Z 692.078,A -85,B 0,C 180,E1 -23792.765,E2 -23792.765} C_VEL
LIN {X 0,Y 183.105,Z 700.933,A -85,B 0,C 180,E1 -23795.45,E2 -23795.45} C_VEL
LIN {X 0,Y 188.436,Z 711.608,A -85,B 0,C 180,E1 -23798.092,E2 -23798.092} C_VEL
LIN {X 0,Y 193.674,Z 723.502,A -85,B 0,C 180,E1 -23800.499,E2 -23800.499} C_VEL
LIN {X 0,Y 198.296,Z 736.292,A -85,B 0,C 180,E1 -23802.553,E2 -23802.553} C_VEL
LIN {X 0,Y 194.101,Z 800.242,A -85,B 0,C 180,E1 -23804.625,E2 -23804.625} C_VEL
LIN {X 0,Y 192.277,Z 814.268,A -85,B 0,C 180,E1 -23805.374,E2 -23805.374} C_VEL
LIN {X 0,Y 189.71,Z 827.37,A -85,B 0,C 180,E1 -23806.371,E2 -23806.371} C_VEL
LIN {X 0,Y 186.662,Z 839.91,A -85,B 0,C 180,E1 -23807.7,E2 -23807.7} C_VEL
LIN {X 0,Y 183.115,Z 851.91,A -85,B 0,C 180,E1 -23809.362,E2 -23809.362} C_VEL
LIN {X 0,Y 180.93,Z 856.995,A -85,B 0,C 180,E1 -23810.083,E2 -23810.083} C_VEL
LIN {X 0,Y 175.776,Z 864.921,A -85,B 0,C 180,E1 -23811.091,E2 -23811.091} C_VEL
LIN {X 0,Y 170.471,Z 872.421,A -85,B 0,C 180,E1 -23812.274,E2 -23812.274} C_VEL
LIN {X 0,Y 168.012,Z 876.783,A -85,B 0,C 180,E1 -23813.297,E2 -23813.297} C_VEL
LIN {X 0,Y 163.921,Z 885.897,A -85,B 0,C 180,E1 -23816.126,E2 -23816.126} C_VEL
LIN {X 0,Y 159.677,Z 894.798,A -85,B 0,C 180,E1 -23819.591,E2 -23819.591} C_VEL
LIN {X 0,Y 156.083,Z 902.204,A -85,B 0,C 180,E1 -23823.238,E2 -23823.238} C_VEL
LIN {X 0,Y 152.916,Z 908.762,A -85,B 0,C 180,E1 -23827.309,E2 -23827.309} C_VEL
LIN {X 0,Y 150.281,Z 914.935,A -85,B 0,C 180,E1 -23832.303,E2 -23832.303} C_VEL
LIN {X 0,Y 148.461,Z 919.828,A -85,B 0,C 180,E1 -23837.7,E2 -23837.7} C_VEL
LIN {X 0,Y 147.835,Z 922.475,A -85,B 0,C 180,E1 -23841.8,E2 -23841.8} C_VEL
LIN {X 0,Y 147.714,Z 924.775,A -85,B 0,C 180,E1 -23847.273,E2 -23847.273} C_VEL
LIN {X 0,Y 147.833,Z 925.405,A -85,B 0,C 180,E1 -23850,E2 -23850} C_VEL
LIN {X 0,Y 147.673,Z 925.618,A -85,B 0,C 180,E1 -23855.462,E2 -23855.462} C_VEL
LIN {X 0,Y 148.219,Z 924.496,A -85,B 0,C 180,E1 -23860.933,E2 -23860.933} C_VEL
LIN {X 0,Y 149.773,Z 922.036,A -85,B 0,C 180,E1 -23866.352,E2 -23866.352} C_VEL
LIN {X 0,Y 152.659,Z 918.187,A -85,B 0,C 180,E1 -23871.61,E2 -23871.61} C_VEL
LIN {X 0,Y 156.568,Z 912.809,A -85,B 0,C 180,E1 -23876.671,E2 -23876.671} C_VEL
LIN {X 0,Y 160.315,Z 907.662,A -85,B 0,C 180,E1 -23880.274,E2 -23880.274} C_VEL
LIN {X 0,Y 165.438,Z 900.333,A -85,B 0,C 180,E1 -23884.255,E2 -23884.255} C_VEL
LIN {X 0,Y 171.506,Z 891.273,A -85,B 0,C 180,E1 -23887.928,E2 -23887.928} C_VEL
LIN {X 0,Y 177.554,Z 881.05,A -85,B 0,C 180,E1 -23891.091,E2 -23891.091} C_VEL
LIN {X 0,Y 183.184,Z 870.261,A -85,B 0,C 180,E1 -23893.676,E2 -23893.676} C_VEL
LIN {X 0,Y 188.663,Z 858.504,A -85,B 0,C 180,E1 -23895.815,E2 -23895.815} C_VEL
LIN {X 0,Y 193.837,Z 845.432,A -85,B 0,C 180,E1 -23897.624,E2 -23897.624} C_VEL
LIN {X 0,Y 197.997,Z 832.557,A -85,B 0,C 180,E1 -23898.962,E2 -23898.962} C_VEL
LIN {X 0,Y 201.375,Z 819.379,A -85,B 0,C 180,E1 -23899.962,E2 -23899.962} C_VEL
LIN {X 0,Y 203.944,Z 805.324,A -85,B 0,C 180,E1 -23900.718,E2 -23900.718} C_VEL
LIN {X 0,Y 205.585,Z 790.042,A -85,B 0,C 180,E1 -23901.244,E2 -23901.244} C_VEL
LIN {X 0,Y 208.537,Z 750.747,A -85,B 0,C 180,E1 -23902.392,E2 -23902.392} C_VEL
LIN {X 0,Y 204.421,Z 740.296,A -85,B 0,C 180,E1 -23904.691,E2 -23904.691} C_VEL
LIN {X 0,Y 199.731,Z 729.824,A -85,B 0,C 180,E1 -23907.526,E2 -23907.526} C_VEL
LIN {X 0,Y 195.716,Z 721.861,A -85,B 0,C 180,E1 -23910.206,E2 -23910.206} C_VEL
LIN {X 0,Y 191.991,Z 714.891,A -85,B 0,C 180,E1 -23913.006,E2 -23913.006} C_VEL
LIN {X 0,Y 188.854,Z 709.488,A -85,B 0,C 180,E1 -23915.672,E2 -23915.672} C_VEL
LIN {X 0,Y 186.249,Z 705.797,A -85,B 0,C 180,E1 -23918.134,E2 -23918.134} C_VEL
LIN {X 0,Y 183.565,Z 702.096,A -85,B 0,C 180,E1 -23921.108,E2 -23921.108} C_VEL
LIN {X 0,Y 182.782,Z 701.088,A -85,B 0,C 180,E1 -23922.086,E2 -23922.086} C_VEL
LIN {X 0,Y 180.354,Z 698.181,A -85,B 0,C 180,E1 -23925.626,E2 -23925.626} C_VEL
LIN {X 0,Y 179.402,Z 696.174,A -85,B 0,C 180,E1 -23927.558,E2 -23927.558} C_VEL
LIN {X 0,Y 176.888,Z 694.016,A -85,B 0,C 180,E1 -23936.014,E2 -23936.014} C_VEL
LIN {X 0,Y 176.987,Z 693.595,A -85,B 0,C 180,E1 -23940.001,E2 -23940.001} C_VEL
LIN {X 0,Y 179.618,Z 696.384,A -85,B 0,C 180,E1 -23948.438,E2 -23948.438} C_VEL
LIN {X 0,Y 181.366,Z 699.689,A -85,B 0,C 180,E1 -23951.597,E2 -23951.597} C_VEL
LIN {X 0,Y 183.373,Z 701.688,A -85,B 0,C 180,E1 -23954.214,E2 -23954.214} C_VEL
LIN {X 0,Y 185.634,Z 705.15,A -85,B 0,C 180,E1 -23956.833,E2 -23956.833} C_VEL
LIN {X 0,Y 187.023,Z 706.805,A -85,B 0,C 180,E1 -23958.203,E2 -23958.203} C_VEL
LIN {X 0,Y 190.616,Z 711.958,A -85,B 0,C 180,E1 -23961.397,E2 -23961.397} C_VEL
LIN {X 0,Y 193.943,Z 716.852,A -85,B 0,C 180,E1 -23963.949,E2 -23963.949} C_VEL
LIN {X 0,Y 198.559,Z 724.092,A -85,B 0,C 180,E1 -23967.058,E2 -23967.058} C_VEL
LIN {X 0,Y 203.411,Z 732.318,A -85,B 0,C 180,E1 -23969.937,E2 -23969.937} C_VEL
LIN {X 0,Y 208.99,Z 742.976,A -85,B 0,C 180,E1 -23972.909,E2 -23972.909} C_VEL
LIN {X 0,Y 207.162,Z 767.807,A -85,B 0,C 180,E1 -23973.649,E2 -23973.649} C_VEL
LIN {X 0,Y 205.283,Z 791.237,A -85,B 0,C 180,E1 -23974.404,E2 -23974.404} C_VEL
LIN {X 0,Y 203.022,Z 805.774,A -85,B 0,C 180,E1 -23975.133,E2 -23975.133} C_VEL
LIN {X 0,Y 200.125,Z 819.02,A -85,B 0,C 180,E1 -23976.127,E2 -23976.127} C_VEL
LIN {X 0,Y 196.521,Z 831.123,A -85,B 0,C 180,E1 -23977.278,E2 -23977.278} C_VEL
LIN {X 0,Y 191.907,Z 844.273,A -85,B 0,C 180,E1 -23979.015,E2 -23979.015} C_VEL
LIN {X 0,Y 187.169,Z 855.467,A -85,B 0,C 180,E1 -23980.916,E2 -23980.916} C_VEL
LIN {X 0,Y 182.464,Z 865.082,A -85,B 0,C 180,E1 -23982.96,E2 -23982.96} C_VEL
LIN {X 0,Y 177.123,Z 874.825,A -85,B 0,C 180,E1 -23985.58,E2 -23985.58} C_VEL
LIN {X 0,Y 172.138,Z 883.144,A -85,B 0,C 180,E1 -23988.437,E2 -23988.437} C_VEL
LIN {X 0,Y 166.293,Z 891.762,A -85,B 0,C 180,E1 -23992.207,E2 -23992.207} C_VEL
LIN {X 0,Y 161.905,Z 897.783,A -85,B 0,C 180,E1 -23995.646,E2 -23995.646} C_VEL
LIN {X 0,Y 156.929,Z 904.164,A -85,B 0,C 180,E1 -24000.487,E2 -24000.487} C_VEL
LIN {X 0,Y 153.088,Z 908.893,A -85,B 0,C 180,E1 -24005.596,E2 -24005.596} C_VEL
LIN {X 0,Y 150.286,Z 912.105,A -85,B 0,C 180,E1 -24010.892,E2 -24010.892} C_VEL
LIN {X 0,Y 148.509,Z 913.91,A -85,B 0,C 180,E1 -24016.313,E2 -24016.313} C_VEL
LIN {X 0,Y 147.81,Z 914.381,A -85,B 0,C 180,E1 -24021.799,E2 -24021.799} C_VEL
LIN {X 0,Y 147.798,Z 913.546,A -85,B 0,C 180,E1 -24027.275,E2 -24027.275} C_VEL
LIN {X 0,Y 148.309,Z 911.405,A -85,B 0,C 180,E1 -24032.716,E2 -24032.716} C_VEL
LIN {X 0,Y 149.637,Z 907.897,A -85,B 0,C 180,E1 -24038.1,E2 -24038.1} C_VEL
LIN {X 0,Y 152.033,Z 902.908,A -85,B 0,C 180,E1 -24043.364,E2 -24043.364} C_VEL
LIN {X 0,Y 154.353,Z 898.088,A -85,B 0,C 180,E1 -24047.215,E2 -24047.215} C_VEL
LIN {X 0,Y 157.713,Z 891.158,A -85,B 0,C 180,E1 -24051.57,E2 -24051.57} C_VEL
LIN {X 0,Y 161.381,Z 883.903,A -85,B 0,C 180,E1 -24055.126,E2 -24055.126} C_VEL
LIN {X 0,Y 165.687,Z 875.171,A -85,B 0,C 180,E1 -24058.503,E2 -24058.503} C_VEL
LIN {X 0,Y 170.347,Z 864.609,A -85,B 0,C 180,E1 -24061.738,E2 -24061.738} C_VEL
LIN {X 0,Y 174.465,Z 853.951,A -85,B 0,C 180,E1 -24064.331,E2 -24064.331} C_VEL
LIN {X 0,Y 177.971,Z 843.715,A -85,B 0,C 180,E1 -24066.324,E2 -24066.324} C_VEL
LIN {X 0,Y 181.738,Z 831.205,A -85,B 0,C 180,E1 -24068.224,E2 -24068.224} C_VEL
LIN {X 0,Y 185.031,Z 818.279,A -85,B 0,C 180,E1 -24069.687,E2 -24069.687} C_VEL
LIN {X 0,Y 187.562,Z 804.42,A -85,B 0,C 180,E1 -24070.887,E2 -24070.887} C_VEL
LIN {X 0,Y 189.414,Z 789.912,A -85,B 0,C 180,E1 -24071.725,E2 -24071.725} C_VEL
LIN {X 0,Y 193.573,Z 731.217,A -85,B 0,C 180,E1 -24073.617,E2 -24073.617} C_VEL
LIN {X 0,Y 193.437,Z 729.842,A -85,B 0,C 180,E1 -24073.732,E2 -24073.732} C_VEL
LIN {X 0,Y 187.789,Z 718.5,A -85,B 0,C 180,E1 -24076.236,E2 -24076.236} C_VEL
LIN {X 0,Y 182.298,Z 708.901,A -85,B 0,C 180,E1 -24078.868,E2 -24078.868} C_VEL
LIN {X 0,Y 176.509,Z 699.764,A -85,B 0,C 180,E1 -24081.948,E2 -24081.948} C_VEL
LIN {X 0,Y 170.824,Z 691.594,A -85,B 0,C 180,E1 -24085.384,E2 -24085.384} C_VEL
LIN {X 0,Y 167.412,Z 687.044,A -85,B 0,C 180,E1 -24087.712,E2 -24087.712} C_VEL
LIN {X 0,Y 164.761,Z 683.569,A -85,B 0,C 180,E1 -24089.709,E2 -24089.709} C_VEL
LIN {X 0,Y 163.821,Z 682.419,A -85,B 0,C 180,E1 -24090.46,E2 -24090.46} C_VEL
LIN {X 0,Y 161.156,Z 679.494,A -85,B 0,C 180,E1 -24092.717,E2 -24092.717} C_VEL
LIN {X 0,Y 159.932,Z 677.418,A -85,B 0,C 180,E1 -24093.931,E2 -24093.931} C_VEL
LIN {X 0,Y 157.09,Z 675.055,A -85,B 0,C 180,E1 -24096.779,E2 -24096.779} C_VEL
LIN {X 0,Y 155.707,Z 672.362,A -85,B 0,C 180,E1 -24098.572,E2 -24098.572} C_VEL
LIN {X 0,Y 155.556,Z 671.852,A -85,B 0,C 180,E1 -24098.811,E2 -24098.811} C_VEL
LIN {X 0,Y 152.532,Z 670.19,A -85,B 0,C 180,E1 -24102.918,E2 -24102.918} C_VEL
LIN {X 0,Y 150.804,Z 667.46,A -85,B 0,C 180,E1 -24106.439,E2 -24106.439} C_VEL
LIN {X 0,Y 150.502,Z 665.845,A -85,B 0,C 180,E1 -24107.629,E2 -24107.629} C_VEL
LIN {X 0,Y 150.686,Z 665.825,A -85,B 0,C 180,E1 -24111.956,E2 -24111.956} C_VEL
LIN {X 0,Y 151.217,Z 665.763,A -85,B 0,C 180,E1 -24119.999,E2 -24119.999} C_VEL
LIN {X 0,Y 150.756,Z 666.025,A -85,B 0,C 180,E1 -24127.617,E2 -24127.617} C_VEL
LIN {X 0,Y 151.244,Z 667.897,A -85,B 0,C 180,E1 -24129.022,E2 -24129.022} C_VEL
LIN {X 0,Y 153.408,Z 670.773,A -85,B 0,C 180,E1 -24132.925,E2 -24132.925} C_VEL
LIN {X 0,Y 155.7,Z 672.055,A -85,B 0,C 180,E1 -24135.881,E2 -24135.881} C_VEL
LIN {X 0,Y 157.121,Z 674.972,A -85,B 0,C 180,E1 -24137.741,E2 -24137.741} C_VEL
LIN {X 0,Y 160.29,Z 677.802,A -85,B 0,C 180,E1 -24140.901,E2 -24140.901} C_VEL
LIN {X 0,Y 162.269,Z 680.928,A -85,B 0,C 180,E1 -24142.773,E2 -24142.773} C_VEL
LIN {X 0,Y 164.467,Z 683.048,A -85,B 0,C 180,E1 -24144.538,E2 -24144.538} C_VEL
LIN {X 0,Y 167.142,Z 686.794,A -85,B 0,C 180,E1 -24146.597,E2 -24146.597} C_VEL
LIN {X 0,Y 168.468,Z 688.39,A -85,B 0,C 180,E1 -24147.525,E2 -24147.525} C_VEL
LIN {X 0,Y 172.225,Z 693.616,A -85,B 0,C 180,E1 -24150.008,E2 -24150.008} C_VEL
LIN {X 0,Y 175.137,Z 697.738,A -85,B 0,C 180,E1 -24151.76,E2 -24151.76} C_VEL
LIN {X 0,Y 179.968,Z 706.689,A -85,B 0,C 180,E1 -24154.531,E2 -24154.531} C_VEL
LIN {X 0,Y 184.759,Z 716.762,A -85,B 0,C 180,E1 -24157.056,E2 -24157.056} C_VEL
LIN {X 0,Y 189.238,Z 727.17,A -85,B 0,C 180,E1 -24159.249,E2 -24159.249} C_VEL
LIN {X 0,Y 193.191,Z 738.26,A -85,B 0,C 180,E1 -24161.13,E2 -24161.13} C_VEL
LIN {X 0,Y 188.939,Z 800.268,A -85,B 0,C 180,E1 -24163.167,E2 -24163.167} C_VEL
LIN {X 0,Y 186.967,Z 814.633,A -85,B 0,C 180,E1 -24163.952,E2 -24163.952} C_VEL
LIN {X 0,Y 184.345,Z 827.495,A -85,B 0,C 180,E1 -24164.953,E2 -24164.953} C_VEL
LIN {X 0,Y 180.921,Z 840.834,A -85,B 0,C 180,E1 -24166.408,E2 -24166.408} C_VEL
LIN {X 0,Y 176.881,Z 853.685,A -85,B 0,C 180,E1 -24168.277,E2 -24168.277} C_VEL
LIN {X 0,Y 172.783,Z 865.089,A -85,B 0,C 180,E1 -24170.445,E2 -24170.445} C_VEL
LIN {X 0,Y 168.752,Z 875.113,A -85,B 0,C 180,E1 -24172.851,E2 -24172.851} C_VEL
LIN {X 0,Y 168.012,Z 876.783,A -85,B 0,C 180,E1 -24173.297,E2 -24173.297} C_VEL
LIN {X 0,Y 165.524,Z 881.081,A -85,B 0,C 180,E1 -24174.402,E2 -24174.402} C_VEL
LIN {X 0,Y 159.943,Z 887.705,A -85,B 0,C 180,E1 -24176.11,E2 -24176.11} C_VEL
LIN {X 0,Y 154.4,Z 893.813,A -85,B 0,C 180,E1 -24178.107,E2 -24178.107} C_VEL
LIN {X 0,Y 152.033,Z 897.297,A -85,B 0,C 180,E1 -24179.651,E2 -24179.651} C_VEL
LIN {X 0,Y 148.036,Z 904.988,A -85,B 0,C 180,E1 -24183.95,E2 -24183.95} C_VEL
LIN {X 0,Y 145.653,Z 909.785,A -85,B 0,C 180,E1 -24187.293,E2 -24187.293} C_VEL
LIN {X 0,Y 143.468,Z 914.542,A -85,B 0,C 180,E1 -24191.433,E2 -24191.433} C_VEL
LIN {X 0,Y 141.484,Z 919.466,A -85,B 0,C 180,E1 -24197.083,E2 -24197.083} C_VEL
LIN {X 0,Y 140.783,Z 922.141,A -85,B 0,C 180,E1 -24201.387,E2 -24201.387} C_VEL
LIN {X 0,Y 140.621,Z 924.469,A -85,B 0,C 180,E1 -24207.135,E2 -24207.135} C_VEL
LIN {X 0,Y 140.736,Z 925.112,A -85,B 0,C 180,E1 -24210,E2 -24210} C_VEL
LIN {X 0,Y 140.599,Z 925.351,A -85,B 0,C 180,E1 -24215.737,E2 -24215.737} C_VEL
LIN {X 0,Y 141.205,Z 924.253,A -85,B 0,C 180,E1 -24221.483,E2 -24221.483} C_VEL
LIN {X 0,Y 142.936,Z 921.82,A -85,B 0,C 180,E1 -24227.158,E2 -24227.158} C_VEL
LIN {X 0,Y 146.047,Z 917.999,A -85,B 0,C 180,E1 -24232.642,E2 -24232.642} C_VEL
LIN {X 0,Y 150.221,Z 912.663,A -85,B 0,C 180,E1 -24237.894,E2 -24237.894} C_VEL
LIN {X 0,Y 154.179,Z 907.534,A -85,B 0,C 180,E1 -24241.615,E2 -24241.615} C_VEL
LIN {X 0,Y 159.601,Z 900.24,A -85,B 0,C 180,E1 -24245.694,E2 -24245.694} C_VEL
LIN {X 0,Y 165.942,Z 891.239,A -85,B 0,C 180,E1 -24249.441,E2 -24249.441} C_VEL
LIN {X 0,Y 171.885,Z 881.717,A -85,B 0,C 180,E1 -24252.47,E2 -24252.47} C_VEL
LIN {X 0,Y 177.567,Z 871.404,A -85,B 0,C 180,E1 -24255.03,E2 -24255.03} C_VEL
LIN {X 0,Y 183.215,Z 859.94,A -85,B 0,C 180,E1 -24257.191,E2 -24257.191} C_VEL
LIN {X 0,Y 188.531,Z 847.253,A -85,B 0,C 180,E1 -24259.014,E2 -24259.014} C_VEL
LIN {X 0,Y 192.805,Z 834.918,A -85,B 0,C 180,E1 -24260.357,E2 -24260.357} C_VEL
LIN {X 0,Y 196.565,Z 821.269,A -85,B 0,C 180,E1 -24261.455,E2 -24261.455} C_VEL
LIN {X 0,Y 199.389,Z 807.227,A -85,B 0,C 180,E1 -24262.253,E2 -24262.253} C_VEL
LIN {X 0,Y 201.208,Z 792.855,A -85,B 0,C 180,E1 -24262.777,E2 -24262.777} C_VEL
LIN {X 0,Y 204.273,Z 753.397,A -85,B 0,C 180,E1 -24263.938,E2 -24263.938} C_VEL
LIN {X 0,Y 200.609,Z 743.813,A -85,B 0,C 180,E1 -24266.156,E2 -24266.156} C_VEL
LIN {X 0,Y 196.179,Z 733.624,A -85,B 0,C 180,E1 -24269.061,E2 -24269.061} C_VEL
LIN {X 0,Y 191.629,Z 724.44,A -85,B 0,C 180,E1 -24272.411,E2 -24272.411} C_VEL
LIN {X 0,Y 189.059,Z 719.664,A -85,B 0,C 180,E1 -24274.544,E2 -24274.544} C_VEL
LIN {X 0,Y 186.838,Z 715.685,A -85,B 0,C 180,E1 -24276.586,E2 -24276.586} C_VEL
LIN {X 0,Y 184.594,Z 712.335,A -85,B 0,C 180,E1 -24278.84,E2 -24278.84} C_VEL
LIN {X 0,Y 181.982,Z 708.511,A -85,B 0,C 180,E1 -24281.923,E2 -24281.923} C_VEL
LIN {X 0,Y 179.034,Z 704.768,A -85,B 0,C 180,E1 -24286.378,E2 -24286.378} C_VEL
LIN {X 0,Y 178.354,Z 703.147,A -85,B 0,C 180,E1 -24287.878,E2 -24287.878} C_VEL
LIN {X 0,Y 175.984,Z 700.915,A -85,B 0,C 180,E1 -24296.741,E2 -24296.741} C_VEL
LIN {X 0,Y 176.174,Z 700.836,A -85,B 0,C 180,E1 -24300.572,E2 -24300.572} C_VEL
LIN {X 0,Y 178.463,Z 703.263,A -85,B 0,C 180,E1 -24307.923,E2 -24307.923} C_VEL
LIN {X 0,Y 180.125,Z 706.503,A -85,B 0,C 180,E1 -24311.099,E2 -24311.099} C_VEL
LIN {X 0,Y 181.952,Z 708.456,A -85,B 0,C 180,E1 -24313.614,E2 -24313.614} C_VEL
LIN {X 0,Y 184.478,Z 712.23,A -85,B 0,C 180,E1 -24316.621,E2 -24316.621} C_VEL
LIN {X 0,Y 185.787,Z 714.109,A -85,B 0,C 180,E1 -24317.972,E2 -24317.972} C_VEL
LIN {X 0,Y 188.707,Z 718.346,A -85,B 0,C 180,E1 -24320.659,E2 -24320.659} C_VEL
LIN {X 0,Y 192.702,Z 724.414,A -85,B 0,C 180,E1 -24323.825,E2 -24323.825} C_VEL
LIN {X 0,Y 198.273,Z 733.764,A -85,B 0,C 180,E1 -24327.607,E2 -24327.607} C_VEL
LIN {X 0,Y 203.42,Z 743.5,A -85,B 0,C 180,E1 -24330.658,E2 -24330.658} C_VEL
LIN {X 0,Y 204.765,Z 746.196,A -85,B 0,C 180,E1 -24331.4,E2 -24331.4} C_VEL
LIN {X 0,Y 201.188,Z 790.728,A -85,B 0,C 180,E1 -24332.755,E2 -24332.755} C_VEL
LIN {X 0,Y 198.994,Z 804.915,A -85,B 0,C 180,E1 -24333.449,E2 -24333.449} C_VEL
LIN {X 0,Y 195.969,Z 818.45,A -85,B 0,C 180,E1 -24334.427,E2 -24334.427} C_VEL
LIN {X 0,Y 192.272,Z 830.739,A -85,B 0,C 180,E1 -24335.582,E2 -24335.582} C_VEL
LIN {X 0,Y 187.809,Z 843.148,A -85,B 0,C 180,E1 -24337.178,E2 -24337.178} C_VEL
LIN {X 0,Y 182.542,Z 855.302,A -85,B 0,C 180,E1 -24339.211,E2 -24339.211} C_VEL
LIN {X 0,Y 177.641,Z 864.991,A -85,B 0,C 180,E1 -24341.263,E2 -24341.263} C_VEL
LIN {X 0,Y 171.653,Z 875.467,A -85,B 0,C 180,E1 -24344.111,E2 -24344.111} C_VEL
LIN {X 0,Y 165.883,Z 884.52,A -85,B 0,C 180,E1 -24347.322,E2 -24347.322} C_VEL
LIN {X 0,Y 160.659,Z 891.828,A -85,B 0,C 180,E1 -24350.632,E2 -24350.632} C_VEL
LIN {X 0,Y 155.946,Z 897.979,A -85,B 0,C 180,E1 -24354.215,E2 -24354.215} C_VEL
LIN {X 0,Y 150.696,Z 904.307,A -85,B 0,C 180,E1 -24359.136,E2 -24359.136} C_VEL
LIN {X 0,Y 146.559,Z 909.069,A -85,B 0,C 180,E1 -24364.432,E2 -24364.432} C_VEL
LIN {X 0,Y 143.513,Z 912.323,A -85,B 0,C 180,E1 -24369.953,E2 -24369.953} C_VEL
LIN {X 0,Y 141.545,Z 914.164,A -85,B 0,C 180,E1 -24375.626,E2 -24375.626} C_VEL
LIN {X 0,Y 140.75,Z 914.663,A -85,B 0,C 180,E1 -24381.385,E2 -24381.385} C_VEL
LIN {X 0,Y 140.702,Z 913.857,A -85,B 0,C 180,E1 -24387.137,E2 -24387.137} C_VEL
LIN {X 0,Y 141.222,Z 911.745,A -85,B 0,C 180,E1 -24392.853,E2 -24392.853} C_VEL
LIN {X 0,Y 142.638,Z 908.268,A -85,B 0,C 180,E1 -24398.501,E2 -24398.501} C_VEL
LIN {X 0,Y 145.161,Z 903.312,A -85,B 0,C 180,E1 -24404.009,E2 -24404.009} C_VEL
LIN {X 0,Y 147.609,Z 898.528,A -85,B 0,C 180,E1 -24408.028,E2 -24408.028} C_VEL
LIN {X 0,Y 151.156,Z 891.637,A -85,B 0,C 180,E1 -24412.556,E2 -24412.556} C_VEL
LIN {X 0,Y 155.022,Z 884.425,A -85,B 0,C 180,E1 -24416.233,E2 -24416.233} C_VEL
LIN {X 0,Y 159.527,Z 875.744,A -85,B 0,C 180,E1 -24419.711,E2 -24419.711} C_VEL
LIN {X 0,Y 164.376,Z 865.244,A -85,B 0,C 180,E1 -24423.034,E2 -24423.034} C_VEL
LIN {X 0,Y 168.693,Z 854.656,A -85,B 0,C 180,E1 -24425.681,E2 -24425.681} C_VEL
LIN {X 0,Y 171.871,Z 845.928,A -85,B 0,C 180,E1 -24427.464,E2 -24427.464} C_VEL
LIN {X 0,Y 175.765,Z 833.88,A -85,B 0,C 180,E1 -24429.403,E2 -24429.403} C_VEL
LIN {X 0,Y 179.424,Z 820.505,A -85,B 0,C 180,E1 -24431.003,E2 -24431.003} C_VEL
LIN {X 0,Y 182.185,Z 806.573,A -85,B 0,C 180,E1 -24432.274,E2 -24432.274} C_VEL
LIN {X 0,Y 184.248,Z 791.865,A -85,B 0,C 180,E1 -24433.174,E2 -24433.174} C_VEL
LIN {X 0,Y 186.306,Z 764.903,A -85,B 0,C 180,E1 -24434.127,E2 -24434.127} C_VEL
LIN {X 0,Y 188.608,Z 732.708,A -85,B 0,C 180,E1 -24435.149,E2 -24435.149} C_VEL
LIN {X 0,Y 183.346,Z 722.09,A -85,B 0,C 180,E1 -24437.65,E2 -24437.65} C_VEL
LIN {X 0,Y 177.644,Z 711.997,A -85,B 0,C 180,E1 -24440.608,E2 -24440.608} C_VEL
LIN {X 0,Y 172.471,Z 703.9,A -85,B 0,C 180,E1 -24443.591,E2 -24443.591} C_VEL
LIN {X 0,Y 167.689,Z 696.909,A -85,B 0,C 180,E1 -24446.716,E2 -24446.716} C_VEL
LIN {X 0,Y 164.885,Z 693.043,A -85,B 0,C 180,E1 -24448.764,E2 -24448.764} C_VEL
LIN {X 0,Y 161.883,Z 688.879,A -85,B 0,C 180,E1 -24451.207,E2 -24451.207} C_VEL
LIN {X 0,Y 159.293,Z 686.014,A -85,B 0,C 180,E1 -24453.506,E2 -24453.506} C_VEL
LIN {X 0,Y 158.104,Z 684.037,A -85,B 0,C 180,E1 -24454.74,E2 -24454.74} C_VEL
LIN {X 0,Y 155.318,Z 681.425,A -85,B 0,C 180,E1 -24457.73,E2 -24457.73} C_VEL
LIN {X 0,Y 153.909,Z 678.681,A -85,B 0,C 180,E1 -24459.685,E2 -24459.685} C_VEL
LIN {X 0,Y 150.853,Z 676.528,A -85,B 0,C 180,E1 -24464.288,E2 -24464.288} C_VEL
LIN {X 0,Y 149.469,Z 673.723,A -85,B 0,C 180,E1 -24467.611,E2 -24467.611} C_VEL
LIN {X 0,Y 149.225,Z 672.802,A -85,B 0,C 180,E1 -24468.463,E2 -24468.463} C_VEL
LIN {X 0,Y 147.747,Z 671.962,A -85,B 0,C 180,E1 -24479.999,E2 -24479.999} C_VEL
LIN {X 0,Y 149.53,Z 672.961,A -85,B 0,C 180,E1 -24486.832,E2 -24486.832} C_VEL
LIN {X 0,Y 150.342,Z 675.323,A -85,B 0,C 180,E1 -24489.077,E2 -24489.077} C_VEL
LIN {X 0,Y 152.551,Z 677.928,A -85,B 0,C 180,E1 -24492.999,E2 -24492.999} C_VEL
LIN {X 0,Y 154.134,Z 678.896,A -85,B 0,C 180,E1 -24495.114,E2 -24495.114} C_VEL
LIN {X 0,Y 155.757,Z 681.905,A -85,B 0,C 180,E1 -24497.287,E2 -24497.287} C_VEL
LIN {X 0,Y 158.469,Z 684.486,A -85,B 0,C 180,E1 -24500.123,E2 -24500.123} C_VEL
LIN {X 0,Y 160.901,Z 688.013,A -85,B 0,C 180,E1 -24502.469,E2 -24502.469} C_VEL
LIN {X 0,Y 162.437,Z 689.646,A -85,B 0,C 180,E1 -24503.76,E2 -24503.76} C_VEL
LIN {X 0,Y 165.354,Z 693.525,A -85,B 0,C 180,E1 -24506.072,E2 -24506.072} C_VEL
LIN {X 0,Y 169.375,Z 699.283,A -85,B 0,C 180,E1 -24508.924,E2 -24508.924} C_VEL
LIN {X 0,Y 172.236,Z 703.425,A -85,B 0,C 180,E1 -24510.75,E2 -24510.75} C_VEL
LIN {X 0,Y 177.222,Z 713.121,A -85,B 0,C 180,E1 -24513.775,E2 -24513.775} C_VEL
LIN {X 0,Y 182.292,Z 724.523,A -85,B 0,C 180,E1 -24516.588,E2 -24516.588} C_VEL
LIN {X 0,Y 185.616,Z 732.879,A -85,B 0,C 180,E1 -24518.316,E2 -24518.316} C_VEL
LIN {X 0,Y 188.243,Z 740.541,A -85,B 0,C 180,E1 -24519.658,E2 -24519.658} C_VEL
LIN {X 0,Y 183.897,Z 800.435,A -85,B 0,C 180,E1 -24521.639,E2 -24521.639} C_VEL
LIN {X 0,Y 181.912,Z 814.368,A -85,B 0,C 180,E1 -24522.41,E2 -24522.41} C_VEL
LIN {X 0,Y 179.1,Z 827.619,A -85,B 0,C 180,E1 -24523.452,E2 -24523.452} C_VEL
LIN {X 0,Y 175.836,Z 839.986,A -85,B 0,C 180,E1 -24524.809,E2 -24524.809} C_VEL
LIN {X 0,Y 171.626,Z 852.946,A -85,B 0,C 180,E1 -24526.693,E2 -24526.693} C_VEL
LIN {X 0,Y 167.29,Z 864.521,A -85,B 0,C 180,E1 -24528.905,E2 -24528.905} C_VEL
LIN {X 0,Y 163.126,Z 874.521,A -85,B 0,C 180,E1 -24531.339,E2 -24531.339} C_VEL
LIN {X 0,Y 158.856,Z 883.713,A -85,B 0,C 180,E1 -24534.112,E2 -24534.112} C_VEL
LIN {X 0,Y 154.223,Z 892.929,A -85,B 0,C 180,E1 -24537.625,E2 -24537.625} C_VEL
LIN {X 0,Y 152.033,Z 897.297,A -85,B 0,C 180,E1 -24539.651,E2 -24539.651} C_VEL
LIN {X 0,Y 149.718,Z 900.651,A -85,B 0,C 180,E1 -24541.291,E2 -24541.291} C_VEL
LIN {X 0,Y 144.412,Z 905.648,A -85,B 0,C 180,E1 -24543.914,E2 -24543.914} C_VEL
LIN {X 0,Y 139.34,Z 910.118,A -85,B 0,C 180,E1 -24546.838,E2 -24546.838} C_VEL
LIN {X 0,Y 137.459,Z 912.559,A -85,B 0,C 180,E1 -24548.902,E2 -24548.902} C_VEL
LIN {X 0,Y 135.423,Z 916.823,A -85,B 0,C 180,E1 -24553.415,E2 -24553.415} C_VEL
LIN {X 0,Y 134.194,Z 920.099,A -85,B 0,C 180,E1 -24557.907,E2 -24557.907} C_VEL
LIN {X 0,Y 133.539,Z 923.161,A -85,B 0,C 180,E1 -24563.958,E2 -24563.958} C_VEL
LIN {X 0,Y 133.568,Z 924.598,A -85,B 0,C 180,E1 -24568.643,E2 -24568.643} C_VEL
LIN {X 0,Y 133.558,Z 924.998,A -85,B 0,C 180,E1 -24571.167,E2 -24571.167} C_VEL
LIN {X 0,Y 133.522,Z 925.083,A -85,B 0,C 180,E1 -24576.042,E2 -24576.042} C_VEL
LIN {X 0,Y 134.219,Z 924.011,A -85,B 0,C 180,E1 -24582.09,E2 -24582.09} C_VEL
LIN {X 0,Y 136.136,Z 921.604,A -85,B 0,C 180,E1 -24588.044,E2 -24588.044} C_VEL
LIN {X 0,Y 139.482,Z 917.811,A -85,B 0,C 180,E1 -24593.771,E2 -24593.771} C_VEL
LIN {X 0,Y 143.939,Z 912.512,A -85,B 0,C 180,E1 -24599.226,E2 -24599.226} C_VEL
LIN {X 0,Y 148.134,Z 907.406,A -85,B 0,C 180,E1 -24603.065,E2 -24603.065} C_VEL
LIN {X 0,Y 153.867,Z 900.148,A -85,B 0,C 180,E1 -24607.243,E2 -24607.243} C_VEL
LIN {X 0,Y 160.504,Z 891.201,A -85,B 0,C 180,E1 -24611.057,E2 -24611.057} C_VEL
LIN {X 0,Y 166.329,Z 882.352,A -85,B 0,C 180,E1 -24613.944,E2 -24613.944} C_VEL
LIN {X 0,Y 172.624,Z 871.482,A -85,B 0,C 180,E1 -24616.697,E2 -24616.697} C_VEL
LIN {X 0,Y 178.472,Z 860.092,A -85,B 0,C 180,E1 -24618.861,E2 -24618.861} C_VEL
LIN {X 0,Y 183.969,Z 847.5,A -85,B 0,C 180,E1 -24620.677,E2 -24620.677} C_VEL
LIN {X 0,Y 188.371,Z 835.299,A -85,B 0,C 180,E1 -24622.014,E2 -24622.014} C_VEL
LIN {X 0,Y 192.244,Z 821.851,A -85,B 0,C 180,E1 -24623.101,E2 -24623.101} C_VEL
LIN {X 0,Y 195.324,Z 807.204,A -85,B 0,C 180,E1 -24623.935,E2 -24623.935} C_VEL
LIN {X 0,Y 197.206,Z 792.821,A -85,B 0,C 180,E1 -24624.463,E2 -24624.463} C_VEL
LIN {X 0,Y 200.206,Z 756.121,A -85,B 0,C 180,E1 -24625.526,E2 -24625.526} C_VEL
LIN {X 0,Y 196.972,Z 747.534,A -85,B 0,C 180,E1 -24627.643,E2 -24627.643} C_VEL
LIN {X 0,Y 193.255,Z 738.691,A -85,B 0,C 180,E1 -24630.276,E2 -24630.276} C_VEL
LIN {X 0,Y 189.011,Z 729.708,A -85,B 0,C 180,E1 -24633.649,E2 -24633.649} C_VEL
LIN {X 0,Y 186.232,Z 724.291,A -85,B 0,C 180,E1 -24636.173,E2 -24636.173} C_VEL
LIN {X 0,Y 184.554,Z 721.351,A -85,B 0,C 180,E1 -24637.846,E2 -24637.846} C_VEL
LIN {X 0,Y 182.789,Z 718.659,A -85,B 0,C 180,E1 -24639.755,E2 -24639.755} C_VEL
LIN {X 0,Y 180.331,Z 714.832,A -85,B 0,C 180,E1 -24642.888,E2 -24642.888} C_VEL
LIN {X 0,Y 177.941,Z 711.762,A -85,B 0,C 180,E1 -24646.729,E2 -24646.729} C_VEL
LIN {X 0,Y 177.139,Z 710.032,A -85,B 0,C 180,E1 -24648.559,E2 -24648.559} C_VEL
LIN {X 0,Y 175.108,Z 707.9,A -85,B 0,C 180,E1 -24657.125,E2 -24657.125} C_VEL
LIN {X 0,Y 175.3,Z 707.942,A -85,B 0,C 180,E1 -24660.575,E2 -24660.575} C_VEL
LIN {X 0,Y 177.324,Z 710.131,A -85,B 0,C 180,E1 -24667.402,E2 -24667.402} C_VEL
LIN {X 0,Y 178.973,Z 713.393,A -85,B 0,C 180,E1 -24670.713,E2 -24670.713} C_VEL
LIN {X 0,Y 180.621,Z 715.305,A -85,B 0,C 180,E1 -24673.099,E2 -24673.099} C_VEL
LIN {X 0,Y 183.097,Z 719.012,A -85,B 0,C 180,E1 -24676.159,E2 -24676.159} C_VEL
LIN {X 0,Y 186.784,Z 724.69,A -85,B 0,C 180,E1 -24679.866,E2 -24679.866} C_VEL
LIN {X 0,Y 190.151,Z 730.011,A -85,B 0,C 180,E1 -24682.706,E2 -24682.706} C_VEL
LIN {X 0,Y 194.807,Z 738.019,A -85,B 0,C 180,E1 -24686.11,E2 -24686.11} C_VEL
LIN {X 0,Y 199.493,Z 747.031,A -85,B 0,C 180,E1 -24689.119,E2 -24689.119} C_VEL
LIN {X 0,Y 200.637,Z 749.382,A -85,B 0,C 180,E1 -24689.804,E2 -24689.804} C_VEL
LIN {X 0,Y 197.182,Z 790.952,A -85,B 0,C 180,E1 -24691.076,E2 -24691.076} C_VEL
LIN {X 0,Y 194.822,Z 805.591,A -85,B 0,C 180,E1 -24691.789,E2 -24691.789} C_VEL
LIN {X 0,Y 191.701,Z 819.022,A -85,B 0,C 180,E1 -24692.763,E2 -24692.763} C_VEL
LIN {X 0,Y 187.582,Z 832.135,A -85,B 0,C 180,E1 -24694.01,E2 -24694.01} C_VEL
LIN {X 0,Y 182.611,Z 845.239,A -85,B 0,C 180,E1 -24695.75,E2 -24695.75} C_VEL
LIN {X 0,Y 176.951,Z 857.499,A -85,B 0,C 180,E1 -24697.873,E2 -24697.873} C_VEL
LIN {X 0,Y 171.894,Z 866.862,A -85,B 0,C 180,E1 -24699.95,E2 -24699.95} C_VEL
LIN {X 0,Y 165.525,Z 877.387,A -85,B 0,C 180,E1 -24702.954,E2 -24702.954} C_VEL
LIN {X 0,Y 159.73,Z 885.898,A -85,B 0,C 180,E1 -24706.133,E2 -24706.133} C_VEL
LIN {X 0,Y 153.466,Z 894.083,A -85,B 0,C 180,E1 -24710.124,E2 -24710.124} C_VEL
LIN {X 0,Y 148.476,Z 900.069,A -85,B 0,C 180,E1 -24713.979,E2 -24713.979} C_VEL
LIN {X 0,Y 143.336,Z 905.812,A -85,B 0,C 180,E1 -24719.014,E2 -24719.014} C_VEL
LIN {X 0,Y 140.104,Z 909.245,A -85,B 0,C 180,E1 -24723.163,E2 -24723.163} C_VEL
LIN {X 0,Y 136.787,Z 912.535,A -85,B 0,C 180,E1 -24728.921,E2 -24728.921} C_VEL
LIN {X 0,Y 134.604,Z 914.416,A -85,B 0,C 180,E1 -24734.867,E2 -24734.867} C_VEL
LIN {X 0,Y 133.686,Z 914.946,A -85,B 0,C 180,E1 -24740.926,E2 -24740.926} C_VEL
LIN {X 0,Y 133.605,Z 914.167,A -85,B 0,C 180,E1 -24746.985,E2 -24746.985} C_VEL
LIN {X 0,Y 134.139,Z 912.085,A -85,B 0,C 180,E1 -24753.004,E2 -24753.004} C_VEL
LIN {X 0,Y 135.629,Z 908.639,A -85,B 0,C 180,E1 -24758.943,E2 -24758.943} C_VEL
LIN {X 0,Y 138.31,Z 903.716,A -85,B 0,C 180,E1 -24764.719,E2 -24764.719} C_VEL
LIN {X 0,Y 141.9,Z 897.178,A -85,B 0,C 180,E1 -24770.286,E2 -24770.286} C_VEL
LIN {X 0,Y 145.898,Z 889.905,A -85,B 0,C 180,E1 -24774.929,E2 -24774.929} C_VEL
LIN {X 0,Y 150.252,Z 882.259,A -85,B 0,C 180,E1 -24778.649,E2 -24778.649} C_VEL
LIN {X 0,Y 155.072,Z 873.091,A -85,B 0,C 180,E1 -24782.176,E2 -24782.176} C_VEL
LIN {X 0,Y 159.375,Z 863.945,A -85,B 0,C 180,E1 -24784.978,E2 -24784.978} C_VEL
LIN {X 0,Y 163.84,Z 853.05,A -85,B 0,C 180,E1 -24787.681,E2 -24787.681} C_VEL
LIN {X 0,Y 168.384,Z 841.057,A -85,B 0,C 180,E1 -24789.921,E2 -24789.921} C_VEL
LIN {X 0,Y 171.978,Z 829.542,A -85,B 0,C 180,E1 -24791.611,E2 -24791.611} C_VEL
LIN {X 0,Y 175.458,Z 815.973,A -85,B 0,C 180,E1 -24793.114,E2 -24793.114} C_VEL
LIN {X 0,Y 178.011,Z 802.539,A -85,B 0,C 180,E1 -24794.194,E2 -24794.194} C_VEL
LIN {X 0,Y 179.831,Z 787.822,A -85,B 0,C 180,E1 -24794.985,E2 -24794.985} C_VEL
LIN {X 0,Y 183.691,Z 735.316,A -85,B 0,C 180,E1 -24796.73,E2 -24796.73} C_VEL
LIN {X 0,Y 179.061,Z 725.775,A -85,B 0,C 180,E1 -24799.111,E2 -24799.111} C_VEL
LIN {X 0,Y 173.834,Z 716.417,A -85,B 0,C 180,E1 -24802.028,E2 -24802.028} C_VEL
LIN {X 0,Y 168.302,Z 707.531,A -85,B 0,C 180,E1 -24805.505,E2 -24805.505} C_VEL
LIN {X 0,Y 163.068,Z 699.712,A -85,B 0,C 180,E1 -24809.344,E2 -24809.344} C_VEL
LIN {X 0,Y 160.198,Z 695.735,A -85,B 0,C 180,E1 -24811.763,E2 -24811.763} C_VEL
LIN {X 0,Y 157.117,Z 691.941,A -85,B 0,C 180,E1 -24814.683,E2 -24814.683} C_VEL
LIN {X 0,Y 156.122,Z 690.496,A -85,B 0,C 180,E1 -24815.761,E2 -24815.761} C_VEL
LIN {X 0,Y 153.454,Z 687.615,A -85,B 0,C 180,E1 -24818.879,E2 -24818.879} C_VEL
LIN {X 0,Y 152.364,Z 685.466,A -85,B 0,C 180,E1 -24820.504,E2 -24820.504} C_VEL
LIN {X 0,Y 149.52,Z 683.15,A -85,B 0,C 180,E1 -24825.147,E2 -24825.147} C_VEL
LIN {X 0,Y 148.258,Z 680.276,A -85,B 0,C 180,E1 -24828.558,E2 -24828.558} C_VEL
LIN {X 0,Y 148.127,Z 679.786,A -85,B 0,C 180,E1 -24829.059,E2 -24829.059} C_VEL
LIN {X 0,Y 146.879,Z 679.021,A -85,B 0,C 180,E1 -24839.999,E2 -24839.999} C_VEL
LIN {X 0,Y 148.388,Z 679.935,A -85,B 0,C 180,E1 -24846.181,E2 -24846.181} C_VEL
LIN {X 0,Y 149.542,Z 682.814,A -85,B 0,C 180,E1 -24849.331,E2 -24849.331} C_VEL
LIN {X 0,Y 151.907,Z 685.201,A -85,B 0,C 180,E1 -24853.374,E2 -24853.374} C_VEL
LIN {X 0,Y 152.691,Z 685.889,A -85,B 0,C 180,E1 -24854.472,E2 -24854.472} C_VEL
LIN {X 0,Y 154.635,Z 689.065,A -85,B 0,C 180,E1 -24857.097,E2 -24857.097} C_VEL
LIN {X 0,Y 156.663,Z 691.099,A -85,B 0,C 180,E1 -24859.307,E2 -24859.307} C_VEL
LIN {X 0,Y 159.502,Z 695.002,A -85,B 0,C 180,E1 -24862.122,E2 -24862.122} C_VEL
LIN {X 0,Y 160.686,Z 696.578,A -85,B 0,C 180,E1 -24863.18,E2 -24863.18} C_VEL
LIN {X 0,Y 163.997,Z 701.176,A -85,B 0,C 180,E1 -24865.89,E2 -24865.89} C_VEL
LIN {X 0,Y 166.952,Z 705.518,A -85,B 0,C 180,E1 -24868.063,E2 -24868.063} C_VEL
LIN {X 0,Y 169.46,Z 709.347,A -85,B 0,C 180,E1 -24869.76,E2 -24869.76} C_VEL
LIN {X 0,Y 173.695,Z 717.902,A -85,B 0,C 180,E1 -24872.505,E2 -24872.505} C_VEL
LIN {X 0,Y 179.111,Z 730.583,A -85,B 0,C 180,E1 -24875.708,E2 -24875.708} C_VEL
LIN {X 0,Y 182.866,Z 740.962,A -85,B 0,C 180,E1 -24877.794,E2 -24877.794} C_VEL
LIN {X 0,Y 183.391,Z 742.665,A -85,B 0,C 180,E1 -24878.087,E2 -24878.087} C_VEL
LIN {X 0,Y 179.097,Z 799.624,A -85,B 0,C 180,E1 -24879.974,E2 -24879.974} C_VEL
LIN {X 0,Y 177.027,Z 813.969,A -85,B 0,C 180,E1 -24880.773,E2 -24880.773} C_VEL
LIN {X 0,Y 173.988,Z 827.742,A -85,B 0,C 180,E1 -24881.861,E2 -24881.861} C_VEL
LIN {X 0,Y 170.323,Z 840.911,A -85,B 0,C 180,E1 -24883.343,E2 -24883.343} C_VEL
LIN {X 0,Y 165.967,Z 853.641,A -85,B 0,C 180,E1 -24885.251,E2 -24885.251} C_VEL
LIN {X 0,Y 161.193,Z 865.721,A -85,B 0,C 180,E1 -24887.653,E2 -24887.653} C_VEL
LIN {X 0,Y 156.663,Z 875.895,A -85,B 0,C 180,E1 -24890.263,E2 -24890.263} C_VEL
LIN {X 0,Y 151.412,Z 886.458,A -85,B 0,C 180,E1 -24893.714,E2 -24893.714} C_VEL
LIN {X 0,Y 146.764,Z 895.173,A -85,B 0,C 180,E1 -24897.403,E2 -24897.403} C_VEL
LIN {X 0,Y 142.232,Z 903.527,A -85,B 0,C 180,E1 -24902.003,E2 -24902.003} C_VEL
LIN {X 0,Y 139.038,Z 909.359,A -85,B 0,C 180,E1 -24906.147,E2 -24906.147} C_VEL
LIN {X 0,Y 137.459,Z 912.559,A -85,B 0,C 180,E1 -24908.902,E2 -24908.902} C_VEL
LIN {X 0,Y 135.733,Z 914.881,A -85,B 0,C 180,E1 -24911.063,E2 -24911.063} C_VEL
LIN {X 0,Y 131.473,Z 918.069,A -85,B 0,C 180,E1 -24914.655,E2 -24914.655} C_VEL
LIN {X 0,Y 128.234,Z 920.106,A -85,B 0,C 180,E1 -24917.745,E2 -24917.745} C_VEL
LIN {X 0,Y 126.77,Z 921.405,A -85,B 0,C 180,E1 -24920.268,E2 -24920.268} C_VEL
LIN {X 0,Y 126.587,Z 921.783,A -85,B 0,C 180,E1 -24921.143,E2 -24921.143} C_VEL
LIN {X 0,Y 126.443,Z 923.858,A -85,B 0,C 180,E1 -24926.813,E2 -24926.813} C_VEL
LIN {X 0,Y 126.512,Z 924.631,A -85,B 0,C 180,E1 -24930.715,E2 -24930.715} C_VEL
LIN {X 0,Y 126.439,Z 924.816,A -85,B 0,C 180,E1 -24936.382,E2 -24936.382} C_VEL
LIN {X 0,Y 127.257,Z 923.769,A -85,B 0,C 180,E1 -24942.762,E2 -24942.762} C_VEL
LIN {X 0,Y 129.375,Z 921.389,A -85,B 0,C 180,E1 -24949.022,E2 -24949.022} C_VEL
LIN {X 0,Y 132.976,Z 917.623,A -85,B 0,C 180,E1 -24955.012,E2 -24955.012} C_VEL
LIN {X 0,Y 137.729,Z 912.359,A -85,B 0,C 180,E1 -24960.682,E2 -24960.682} C_VEL
LIN {X 0,Y 142.203,Z 907.281,A -85,B 0,C 180,E1 -24964.635,E2 -24964.635} C_VEL
LIN {X 0,Y 148.236,Z 900.057,A -85,B 0,C 180,E1 -24968.917,E2 -24968.917} C_VEL
LIN {X 0,Y 155.201,Z 891.157,A -85,B 0,C 180,E1 -24972.785,E2 -24972.785} C_VEL
LIN {X 0,Y 161.981,Z 881.214,A -85,B 0,C 180,E1 -24976.037,E2 -24976.037} C_VEL
LIN {X 0,Y 168.423,Z 870.492,A -85,B 0,C 180,E1 -24978.686,E2 -24978.686} C_VEL
LIN {X 0,Y 174.513,Z 858.954,A -85,B 0,C 180,E1 -24980.826,E2 -24980.826} C_VEL
LIN {X 0,Y 180.201,Z 846.169,A -85,B 0,C 180,E1 -24982.621,E2 -24982.621} C_VEL
LIN {X 0,Y 184.752,Z 833.697,A -85,B 0,C 180,E1 -24983.935,E2 -24983.935} C_VEL
LIN {X 0,Y 188.759,Z 819.839,A -85,B 0,C 180,E1 -24984.997,E2 -24984.997} C_VEL
LIN {X 0,Y 191.73,Z 805.524,A -85,B 0,C 180,E1 -24985.769,E2 -24985.769} C_VEL
LIN {X 0,Y 193.492,Z 791.567,A -85,B 0,C 180,E1 -24986.258,E2 -24986.258} C_VEL
LIN {X 0,Y 196.251,Z 758.789,A -85,B 0,C 180,E1 -24987.205,E2 -24987.205} C_VEL
LIN {X 0,Y 192.25,Z 748.11,A -85,B 0,C 180,E1 -24990.104,E2 -24990.104} C_VEL
LIN {X 0,Y 188.805,Z 740.036,A -85,B 0,C 180,E1 -24992.862,E2 -24992.862} C_VEL
LIN {X 0,Y 185.478,Z 732.806,A -85,B 0,C 180,E1 -24995.886,E2 -24995.886} C_VEL
LIN {X 0,Y 183.119,Z 728.261,A -85,B 0,C 180,E1 -24998.307,E2 -24998.307} C_VEL
LIN {X 0,Y 181.226,Z 725.218,A -85,B 0,C 180,E1 -25000.46,E2 -25000.46} C_VEL
LIN {X 0,Y 178.82,Z 721.468,A -85,B 0,C 180,E1 -25003.709,E2 -25003.709} C_VEL
LIN {X 0,Y 176.52,Z 717.984,A -85,B 0,C 180,E1 -25007.847,E2 -25007.847} C_VEL
LIN {X 0,Y 176.029,Z 716.953,A -85,B 0,C 180,E1 -25009.069,E2 -25009.069} C_VEL
LIN {X 0,Y 174.24,Z 714.965,A -85,B 0,C 180,E1 -25017.111,E2 -25017.111} C_VEL
LIN {X 0,Y 174.43,Z 715.017,A -85,B 0,C 180,E1 -25020.578,E2 -25020.578} C_VEL
LIN {X 0,Y 176.251,Z 717.15,A -85,B 0,C 180,E1 -25027.015,E2 -25027.015} C_VEL
LIN {X 0,Y 178.032,Z 720.578,A -85,B 0,C 180,E1 -25030.664,E2 -25030.664} C_VEL
LIN {X 0,Y 179.223,Z 722.016,A -85,B 0,C 180,E1 -25032.456,E2 -25032.456} C_VEL
LIN {X 0,Y 182.247,Z 726.804,A -85,B 0,C 180,E1 -25036.308,E2 -25036.308} C_VEL
LIN {X 0,Y 184.805,Z 730.853,A -85,B 0,C 180,E1 -25038.965,E2 -25038.965} C_VEL
LIN {X 0,Y 188.357,Z 736.746,A -85,B 0,C 180,E1 -25042.125,E2 -25042.125} C_VEL
LIN {X 0,Y 193.038,Z 745.22,A -85,B 0,C 180,E1 -25045.689,E2 -25045.689} C_VEL
LIN {X 0,Y 196.674,Z 752.623,A -85,B 0,C 180,E1 -25048.147,E2 -25048.147} C_VEL
LIN {X 0,Y 193.329,Z 791.375,A -85,B 0,C 180,E1 -25049.339,E2 -25049.339} C_VEL
LIN {X 0,Y 190.871,Z 806.062,A -85,B 0,C 180,E1 -25050.049,E2 -25050.049} C_VEL
LIN {X 0,Y 187.609,Z 819.595,A -85,B 0,C 180,E1 -25051.028,E2 -25051.028} C_VEL
LIN {X 0,Y 183.035,Z 833.53,A -85,B 0,C 180,E1 -25052.357,E2 -25052.357} C_VEL
LIN {X 0,Y 178.083,Z 845.985,A -85,B 0,C 180,E1 -25054.029,E2 -25054.029} C_VEL
LIN {X 0,Y 172.65,Z 857.338,A -85,B 0,C 180,E1 -25055.998,E2 -25055.998} C_VEL
LIN {X 0,Y 167.369,Z 866.774,A -85,B 0,C 180,E1 -25058.064,E2 -25058.064} C_VEL
LIN {X 0,Y 161.064,Z 876.783,A -85,B 0,C 180,E1 -25060.884,E2 -25060.884} C_VEL
LIN {X 0,Y 154.619,Z 885.923,A -85,B 0,C 180,E1 -25064.283,E2 -25064.283} C_VEL
LIN {X 0,Y 148.011,Z 894.171,A -85,B 0,C 180,E1 -25068.336,E2 -25068.336} C_VEL
LIN {X 0,Y 143.078,Z 899.778,A -85,B 0,C 180,E1 -25071.992,E2 -25071.992} C_VEL
LIN {X 0,Y 138.536,Z 904.593,A -85,B 0,C 180,E1 -25076.08,E2 -25076.08} C_VEL
LIN {X 0,Y 133.719,Z 909.423,A -85,B 0,C 180,E1 -25081.77,E2 -25081.77} C_VEL
LIN {X 0,Y 130.114,Z 912.744,A -85,B 0,C 180,E1 -25087.784,E2 -25087.784} C_VEL
LIN {X 0,Y 127.688,Z 914.664,A -85,B 0,C 180,E1 -25094.026,E2 -25094.026} C_VEL
LIN {X 0,Y 126.623,Z 915.229,A -85,B 0,C 180,E1 -25100.415,E2 -25100.415} C_VEL
LIN {X 0,Y 126.507,Z 914.478,A -85,B 0,C 180,E1 -25106.816,E2 -25106.816} C_VEL
LIN {X 0,Y 127.059,Z 912.426,A -85,B 0,C 180,E1 -25113.171,E2 -25113.171} C_VEL
LIN {X 0,Y 128.631,Z 909.011,A -85,B 0,C 180,E1 -25119.434,E2 -25119.434} C_VEL
LIN {X 0,Y 131.467,Z 904.121,A -85,B 0,C 180,E1 -25125.503,E2 -25125.503} C_VEL
LIN {X 0,Y 135.296,Z 897.617,A -85,B 0,C 180,E1 -25131.323,E2 -25131.323} C_VEL
LIN {X 0,Y 139.512,Z 890.386,A -85,B 0,C 180,E1 -25136.155,E2 -25136.155} C_VEL
LIN {X 0,Y 144.921,Z 881.376,A -85,B 0,C 180,E1 -25140.611,E2 -25140.611} C_VEL
LIN {X 0,Y 150.04,Z 871.951,A -85,B 0,C 180,E1 -25144.201,E2 -25144.201} C_VEL
LIN {X 0,Y 154.501,Z 862.598,A -85,B 0,C 180,E1 -25147.065,E2 -25147.065} C_VEL
LIN {X 0,Y 158.314,Z 853.752,A -85,B 0,C 180,E1 -25149.242,E2 -25149.242} C_VEL
LIN {X 0,Y 163.042,Z 841.854,A -85,B 0,C 180,E1 -25151.51,E2 -25151.51} C_VEL
LIN {X 0,Y 166.773,Z 830.46,A -85,B 0,C 180,E1 -25153.22,E2 -25153.22} C_VEL
LIN {X 0,Y 170.399,Z 817.111,A -85,B 0,C 180,E1 -25154.728,E2 -25154.728} C_VEL
LIN {X 0,Y 173.166,Z 803.241,A -85,B 0,C 180,E1 -25155.878,E2 -25155.878} C_VEL
LIN {X 0,Y 174.999,Z 789.349,A -85,B 0,C 180,E1 -25156.656,E2 -25156.656} C_VEL
LIN {X 0,Y 179.008,Z 738.105,A -85,B 0,C 180,E1 -25158.351,E2 -25158.351} C_VEL
LIN {X 0,Y 174.792,Z 729.349,A -85,B 0,C 180,E1 -25160.697,E2 -25160.697} C_VEL
LIN {X 0,Y 169.764,Z 720.134,A -85,B 0,C 180,E1 -25163.75,E2 -25163.75} C_VEL
LIN {X 0,Y 164.445,Z 711.604,A -85,B 0,C 180,E1 -25167.405,E2 -25167.405} C_VEL
LIN {X 0,Y 160.68,Z 705.776,A -85,B 0,C 180,E1 -25170.407,E2 -25170.407} C_VEL
LIN {X 0,Y 157.656,Z 701.525,A -85,B 0,C 180,E1 -25173.141,E2 -25173.141} C_VEL
LIN {X 0,Y 154.905,Z 697.717,A -85,B 0,C 180,E1 -25176.01,E2 -25176.01} C_VEL
LIN {X 0,Y 151.646,Z 693.74,A -85,B 0,C 180,E1 -25180.076,E2 -25180.076} C_VEL
LIN {X 0,Y 150.807,Z 692.23,A -85,B 0,C 180,E1 -25181.4,E2 -25181.4} C_VEL
LIN {X 0,Y 148.256,Z 689.83,A -85,B 0,C 180,E1 -25185.939,E2 -25185.939} C_VEL
LIN {X 0,Y 147.125,Z 687,A -85,B 0,C 180,E1 -25189.353,E2 -25189.353} C_VEL
LIN {X 0,Y 146.469,Z 686.549,A -85,B 0,C 180,E1 -25191.723,E2 -25191.723} C_VEL
LIN {X 0,Y 146.011,Z 686.079,A -85,B 0,C 180,E1 -25199.999,E2 -25199.999} C_VEL
LIN {X 0,Y 147.303,Z 686.978,A -85,B 0,C 180,E1 -25205.647,E2 -25205.647} C_VEL
LIN {X 0,Y 148.72,Z 690.2,A -85,B 0,C 180,E1 -25209.52,E2 -25209.52} C_VEL
LIN {X 0,Y 151.206,Z 692.606,A -85,B 0,C 180,E1 -25213.694,E2 -25213.694} C_VEL
LIN {X 0,Y 153.305,Z 695.982,A -85,B 0,C 180,E1 -25216.649,E2 -25216.649} C_VEL
LIN {X 0,Y 154.866,Z 697.607,A -85,B 0,C 180,E1 -25218.436,E2 -25218.436} C_VEL
LIN {X 0,Y 157.866,Z 701.74,A -85,B 0,C 180,E1 -25221.547,E2 -25221.547} C_VEL
LIN {X 0,Y 161.667,Z 707.287,A -85,B 0,C 180,E1 -25224.915,E2 -25224.915} C_VEL
LIN {X 0,Y 165.115,Z 712.547,A -85,B 0,C 180,E1 -25227.573,E2 -25227.573} C_VEL
LIN {X 0,Y 167.02,Z 715.81,A -85,B 0,C 180,E1 -25228.94,E2 -25228.94} C_VEL
LIN {X 0,Y 171.014,Z 724.531,A -85,B 0,C 180,E1 -25231.695,E2 -25231.695} C_VEL
LIN {X 0,Y 175.818,Z 736.345,A -85,B 0,C 180,E1 -25234.712,E2 -25234.712} C_VEL
LIN {X 0,Y 178.679,Z 744.767,A -85,B 0,C 180,E1 -25236.429,E2 -25236.429} C_VEL
LIN {X 0,Y 174.334,Z 799.929,A -85,B 0,C 180,E1 -25238.281,E2 -25238.281} C_VEL
LIN {X 0,Y 172.081,Z 814.534,A -85,B 0,C 180,E1 -25239.105,E2 -25239.105} C_VEL
LIN {X 0,Y 169.018,Z 827.857,A -85,B 0,C 180,E1 -25240.176,E2 -25240.176} C_VEL
LIN {X 0,Y 164.928,Z 841.828,A -85,B 0,C 180,E1 -25241.778,E2 -25241.778} C_VEL
LIN {X 0,Y 160.42,Z 854.331,A -85,B 0,C 180,E1 -25243.708,E2 -25243.708} C_VEL
LIN {X 0,Y 155.668,Z 865.773,A -85,B 0,C 180,E1 -25246.042,E2 -25246.042} C_VEL
LIN {X 0,Y 151.191,Z 875.413,A -85,B 0,C 180,E1 -25248.568,E2 -25248.568} C_VEL
LIN {X 0,Y 145.718,Z 885.916,A -85,B 0,C 180,E1 -25252.052,E2 -25252.052} C_VEL
LIN {X 0,Y 140.783,Z 894.675,A -85,B 0,C 180,E1 -25255.832,E2 -25255.832} C_VEL
LIN {X 0,Y 135.944,Z 903.081,A -85,B 0,C 180,E1 -25260.585,E2 -25260.585} C_VEL
LIN {X 0,Y 132.471,Z 908.932,A -85,B 0,C 180,E1 -25264.885,E2 -25264.885} C_VEL
LIN {X 0,Y 129.958,Z 913.758,A -85,B 0,C 180,E1 -25269.42,E2 -25269.42} C_VEL
LIN {X 0,Y 127.568,Z 918.741,A -85,B 0,C 180,E1 -25275.645,E2 -25275.645} C_VEL
LIN {X 0,Y 126.587,Z 921.783,A -85,B 0,C 180,E1 -25281.143,E2 -25281.143} C_VEL
LIN {X 0,Y 126.121,Z 922.571,A -85,B 0,C 180,E1 -25282.891,E2 -25282.891} C_VEL
LIN {X 0,Y 124.635,Z 923.449,A -85,B 0,C 180,E1 -25285.491,E2 -25285.491} C_VEL
LIN {X 0,Y 120.289,Z 924.51,A -85,B 0,C 180,E1 -25291.726,E2 -25291.726} C_VEL
LIN {X 0,Y 119.332,Z 924.607,A -85,B 0,C 180,E1 -25294.572,E2 -25294.572} C_VEL
LIN {X 0,Y 119.287,Z 924.552,A -85,B 0,C 180,E1 -25295.536,E2 -25295.536} C_VEL
LIN {X 0,Y 119.639,Z 924.202,A -85,B 0,C 180,E1 -25300.15,E2 -25300.15} C_VEL
LIN {X 0,Y 121.237,Z 922.518,A -85,B 0,C 180,E1 -25306.848,E2 -25306.848} C_VEL
LIN {X 0,Y 124.395,Z 919.483,A -85,B 0,C 180,E1 -25313.296,E2 -25313.296} C_VEL
LIN {X 0,Y 128.883,Z 915.012,A -85,B 0,C 180,E1 -25319.391,E2 -25319.391} C_VEL
LIN {X 0,Y 134.725,Z 908.973,A -85,B 0,C 180,E1 -25325.017,E2 -25325.017} C_VEL
LIN {X 0,Y 140.833,Z 902.208,A -85,B 0,C 180,E1 -25329.514,E2 -25329.514} C_VEL
LIN {X 0,Y 147.93,Z 893.821,A -85,B 0,C 180,E1 -25333.541,E2 -25333.541} C_VEL
LIN {X 0,Y 154.483,Z 885.103,A -85,B 0,C 180,E1 -25336.71,E2 -25336.71} C_VEL
LIN {X 0,Y 161.378,Z 874.561,A -85,B 0,C 180,E1 -25339.652,E2 -25339.652} C_VEL
LIN {X 0,Y 168.193,Z 862.779,A -85,B 0,C 180,E1 -25342.064,E2 -25342.064} C_VEL
LIN {X 0,Y 174.018,Z 850.975,A -85,B 0,C 180,E1 -25343.875,E2 -25343.875} C_VEL
LIN {X 0,Y 179.371,Z 837.954,A -85,B 0,C 180,E1 -25345.367,E2 -25345.367} C_VEL
LIN {X 0,Y 183.767,Z 824.311,A -85,B 0,C 180,E1 -25346.532,E2 -25346.532} C_VEL
LIN {X 0,Y 187.261,Z 809.664,A -85,B 0,C 180,E1 -25347.393,E2 -25347.393} C_VEL
LIN {X 0,Y 189.496,Z 795.173,A -85,B 0,C 180,E1 -25347.96,E2 -25347.96} C_VEL
LIN {X 0,Y 192.467,Z 761.526,A -85,B 0,C 180,E1 -25348.951,E2 -25348.951} C_VEL
LIN {X 0,Y 188.883,Z 751.736,A -85,B 0,C 180,E1 -25351.802,E2 -25351.802} C_VEL
LIN {X 0,Y 185.48,Z 743.478,A -85,B 0,C 180,E1 -25354.827,E2 -25354.827} C_VEL
LIN {X 0,Y 182.991,Z 737.932,A -85,B 0,C 180,E1 -25357.333,E2 -25357.333} C_VEL
LIN {X 0,Y 181.273,Z 734.454,A -85,B 0,C 180,E1 -25359.252,E2 -25359.252} C_VEL
LIN {X 0,Y 179.621,Z 731.701,A -85,B 0,C 180,E1 -25361.261,E2 -25361.261} C_VEL
LIN {X 0,Y 177.479,Z 728.202,A -85,B 0,C 180,E1 -25364.35,E2 -25364.35} C_VEL
LIN {X 0,Y 175.312,Z 724.608,A -85,B 0,C 180,E1 -25368.584,E2 -25368.584} C_VEL
LIN {X 0,Y 174.934,Z 723.87,A -85,B 0,C 180,E1 -25369.585,E2 -25369.585} C_VEL
LIN {X 0,Y 173.374,Z 721.913,A -85,B 0,C 180,E1 -25377.677,E2 -25377.677} C_VEL
LIN {X 0,Y 173.529,Z 722.012,A -85,B 0,C 180,E1 -25380.291,E2 -25380.291} C_VEL
LIN {X 0,Y 175.188,Z 724.154,A -85,B 0,C 180,E1 -25386.624,E2 -25386.624} C_VEL
LIN {X 0,Y 176.905,Z 727.5,A -85,B 0,C 180,E1 -25390.299,E2 -25390.299} C_VEL
LIN {X 0,Y 177.868,Z 728.741,A -85,B 0,C 180,E1 -25391.828,E2 -25391.828} C_VEL
LIN {X 0,Y 180.749,Z 733.531,A -85,B 0,C 180,E1 -25395.709,E2 -25395.709} C_VEL
LIN {X 0,Y 183.26,Z 737.732,A -85,B 0,C 180,E1 -25398.446,E2 -25398.446} C_VEL
LIN {X 0,Y 186.274,Z 742.946,A -85,B 0,C 180,E1 -25401.267,E2 -25401.267} C_VEL
LIN {X 0,Y 190.476,Z 750.925,A -85,B 0,C 180,E1 -25404.671,E2 -25404.671} C_VEL
LIN {X 0,Y 192.883,Z 755.977,A -85,B 0,C 180,E1 -25406.43,E2 -25406.43} C_VEL
LIN {X 0,Y 189.648,Z 791.889,A -85,B 0,C 180,E1 -25407.536,E2 -25407.536} C_VEL
LIN {X 0,Y 187.232,Z 805.981,A -85,B 0,C 180,E1 -25408.207,E2 -25408.207} C_VEL
LIN {X 0,Y 183.694,Z 820.175,A -85,B 0,C 180,E1 -25409.216,E2 -25409.216} C_VEL
LIN {X 0,Y 179.313,Z 833.153,A -85,B 0,C 180,E1 -25410.428,E2 -25410.428} C_VEL
LIN {X 0,Y 174.166,Z 845.731,A -85,B 0,C 180,E1 -25412.07,E2 -25412.07} C_VEL
LIN {X 0,Y 168.541,Z 857.177,A -85,B 0,C 180,E1 -25414.028,E2 -25414.028} C_VEL
LIN {X 0,Y 163.046,Z 866.687,A -85,B 0,C 180,E1 -25416.079,E2 -25416.079} C_VEL
LIN {X 0,Y 155.973,Z 877.452,A -85,B 0,C 180,E1 -25419.112,E2 -25419.112} C_VEL
LIN {X 0,Y 149.689,Z 885.947,A -85,B 0,C 180,E1 -25422.314,E2 -25422.314} C_VEL
LIN {X 0,Y 142.704,Z 894.254,A -85,B 0,C 180,E1 -25426.411,E2 -25426.411} C_VEL
LIN {X 0,Y 137.107,Z 900.288,A -85,B 0,C 180,E1 -25430.442,E2 -25430.442} C_VEL
LIN {X 0,Y 131.189,Z 906.133,A -85,B 0,C 180,E1 -25435.771,E2 -25435.771} C_VEL
LIN {X 0,Y 127.415,Z 909.6,A -85,B 0,C 180,E1 -25440.237,E2 -25440.237} C_VEL
LIN {X 0,Y 123.503,Z 912.953,A -85,B 0,C 180,E1 -25446.526,E2 -25446.526} C_VEL
LIN {X 0,Y 120.804,Z 914.907,A -85,B 0,C 180,E1 -25453.089,E2 -25453.089} C_VEL
LIN {X 0,Y 119.585,Z 915.508,A -85,B 0,C 180,E1 -25459.845,E2 -25459.845} C_VEL
LIN {X 0,Y 119.395,Z 914.789,A -85,B 0,C 180,E1 -25466.626,E2 -25466.626} C_VEL
LIN {X 0,Y 119.607,Z 913.941,A -85,B 0,C 180,E1 -25470,E2 -25470} C_VEL
LIN {X 0,Y 120.627,Z 911.25,A -85,B 0,C 180,E1 -25476.692,E2 -25476.692} C_VEL
LIN {X 0,Y 122.987,Z 907.145,A -85,B 0,C 180,E1 -25483.214,E2 -25483.214} C_VEL
LIN {X 0,Y 125.852,Z 902.576,A -85,B 0,C 180,E1 -25488.441,E2 -25488.441} C_VEL
LIN {X 0,Y 129.847,Z 896.15,A -85,B 0,C 180,E1 -25493.95,E2 -25493.95} C_VEL
LIN {X 0,Y 134.713,Z 888.475,A -85,B 0,C 180,E1 -25498.854,E2 -25498.854} C_VEL
LIN {X 0,Y 139.737,Z 880.447,A -85,B 0,C 180,E1 -25502.729,E2 -25502.729} C_VEL
LIN {X 0,Y 145.147,Z 870.788,A -85,B 0,C 180,E1 -25506.381,E2 -25506.381} C_VEL
LIN {X 0,Y 150.477,Z 860.075,A -85,B 0,C 180,E1 -25509.521,E2 -25509.521} C_VEL
LIN {X 0,Y 154.505,Z 850.775,A -85,B 0,C 180,E1 -25511.702,E2 -25511.702} C_VEL
LIN {X 0,Y 159.442,Z 838.084,A -85,B 0,C 180,E1 -25513.967,E2 -25513.967} C_VEL
LIN {X 0,Y 163.462,Z 825.704,A -85,B 0,C 180,E1 -25515.626,E2 -25515.626} C_VEL
LIN {X 0,Y 166.868,Z 811.979,A -85,B 0,C 180,E1 -25517.037,E2 -25517.037} C_VEL
LIN {X 0,Y 169.487,Z 797.596,A -85,B 0,C 180,E1 -25518.057,E2 -25518.057} C_VEL
LIN {X 0,Y 171.111,Z 782.624,A -85,B 0,C 180,E1 -25518.72,E2 -25518.72} C_VEL
LIN {X 0,Y 174.436,Z 740.795,A -85,B 0,C 180,E1 -25520.081,E2 -25520.081} C_VEL
LIN {X 0,Y 169.38,Z 730.465,A -85,B 0,C 180,E1 -25523.171,E2 -25523.171} C_VEL
LIN {X 0,Y 164.762,Z 722.15,A -85,B 0,C 180,E1 -25526.321,E2 -25526.321} C_VEL
LIN {X 0,Y 159.881,Z 714.21,A -85,B 0,C 180,E1 -25530.151,E2 -25530.151} C_VEL
LIN {X 0,Y 157.474,Z 710.601,A -85,B 0,C 180,E1 -25532.305,E2 -25532.305} C_VEL
LIN {X 0,Y 155.656,Z 707.857,A -85,B 0,C 180,E1 -25534.107,E2 -25534.107} C_VEL
LIN {X 0,Y 152.716,Z 703.654,A -85,B 0,C 180,E1 -25537.419,E2 -25537.419} C_VEL
LIN {X 0,Y 150.162,Z 700.377,A -85,B 0,C 180,E1 -25540.875,E2 -25540.875} C_VEL
LIN {X 0,Y 149.426,Z 699.028,A -85,B 0,C 180,E1 -25542.109,E2 -25542.109} C_VEL
LIN {X 0,Y 147.07,Z 696.607,A -85,B 0,C 180,E1 -25546.617,E2 -25546.617} C_VEL
LIN {X 0,Y 145.955,Z 693.705,A -85,B 0,C 180,E1 -25550.382,E2 -25550.382} C_VEL
LIN {X 0,Y 145.232,Z 693.215,A -85,B 0,C 180,E1 -25560.719,E2 -25560.719} C_VEL
LIN {X 0,Y 146.253,Z 694.034,A -85,B 0,C 180,E1 -25565.169,E2 -25565.169} C_VEL
LIN {X 0,Y 147.972,Z 697.63,A -85,B 0,C 180,E1 -25569.846,E2 -25569.846} C_VEL
LIN {X 0,Y 149.806,Z 699.444,A -85,B 0,C 180,E1 -25572.999,E2 -25572.999} C_VEL
LIN {X 0,Y 151.925,Z 702.805,A -85,B 0,C 180,E1 -25576.114,E2 -25576.114} C_VEL
LIN {X 0,Y 153.225,Z 704.307,A -85,B 0,C 180,E1 -25577.689,E2 -25577.689} C_VEL
LIN {X 0,Y 156.623,Z 709.265,A -85,B 0,C 180,E1 -25581.36,E2 -25581.36} C_VEL
LIN {X 0,Y 159.578,Z 713.739,A -85,B 0,C 180,E1 -25584.082,E2 -25584.082} C_VEL
LIN {X 0,Y 163.53,Z 720,A -85,B 0,C 180,E1 -25587.256,E2 -25587.256} C_VEL
LIN {X 0,Y 167.495,Z 728.913,A -85,B 0,C 180,E1 -25590.232,E2 -25590.232} C_VEL
LIN {X 0,Y 172.097,Z 740.818,A -85,B 0,C 180,E1 -25593.368,E2 -25593.368} C_VEL
LIN {X 0,Y 174.1,Z 746.94,A -85,B 0,C 180,E1 -25594.677,E2 -25594.677} C_VEL
LIN {X 0,Y 169.799,Z 799.506,A -85,B 0,C 180,E1 -25596.448,E2 -25596.448} C_VEL
LIN {X 0,Y 167.514,Z 814.014,A -85,B 0,C 180,E1 -25597.266,E2 -25597.266} C_VEL
LIN {X 0,Y 164.205,Z 827.971,A -85,B 0,C 180,E1 -25598.392,E2 -25598.392} C_VEL
LIN {X 0,Y 160.28,Z 840.972,A -85,B 0,C 180,E1 -25599.883,E2 -25599.883} C_VEL
LIN {X 0,Y 155.55,Z 853.58,A -85,B 0,C 180,E1 -25601.798,E2 -25601.798} C_VEL
LIN {X 0,Y 150.6,Z 865.103,A -85,B 0,C 180,E1 -25604.151,E2 -25604.151} C_VEL
LIN {X 0,Y 145.789,Z 875.062,A -85,B 0,C 180,E1 -25606.784,E2 -25606.784} C_VEL
LIN {X 0,Y 140.138,Z 885.37,A -85,B 0,C 180,E1 -25610.251,E2 -25610.251} C_VEL
LIN {X 0,Y 134.912,Z 894.175,A -85,B 0,C 180,E1 -25614.122,E2 -25614.122} C_VEL
LIN {X 0,Y 129.758,Z 902.628,A -85,B 0,C 180,E1 -25619.033,E2 -25619.033} C_VEL
LIN {X 0,Y 125.982,Z 908.504,A -85,B 0,C 180,E1 -25623.494,E2 -25623.494} C_VEL
LIN {X 0,Y 123.277,Z 913.365,A -85,B 0,C 180,E1 -25628.249,E2 -25628.249} C_VEL
LIN {X 0,Y 120.658,Z 918.379,A -85,B 0,C 180,E1 -25634.804,E2 -25634.804} C_VEL
LIN {X 0,Y 119.503,Z 921.611,A -85,B 0,C 180,E1 -25641.006,E2 -25641.006} C_VEL
LIN {X 0,Y 119.353,Z 923.552,A -85,B 0,C 180,E1 -25646.624,E2 -25646.624} C_VEL
LIN {X 0,Y 119.474,Z 924.236,A -85,B 0,C 180,E1 -25650,E2 -25650} C_VEL
LIN {X 0,Y 119.287,Z 924.552,A -85,B 0,C 180,E1 -25655.536,E2 -25655.536} C_VEL
LIN {X 0,Y 119.079,Z 924.499,A -85,B 0,C 180,E1 -25657.424,E2 -25657.424} C_VEL
LIN {X 0,Y 117.567,Z 924.012,A -85,B 0,C 180,E1 -25661.175,E2 -25661.175} C_VEL
LIN {X 0,Y 115.227,Z 922.595,A -85,B 0,C 180,E1 -25666.907,E2 -25666.907} C_VEL
LIN {X 0,Y 115.314,Z 921.611,A -85,B 0,C 180,E1 -25669.817,E2 -25669.817} C_VEL
LIN {X 0,Y 115.68,Z 921.177,A -85,B 0,C 180,E1 -25670.766,E2 -25670.766} C_VEL
LIN {X 0,Y 118.97,Z 918.33,A -85,B 0,C 180,E1 -25676.299,E2 -25676.299} C_VEL
LIN {X 0,Y 124.137,Z 913.484,A -85,B 0,C 180,E1 -25682.536,E2 -25682.536} C_VEL
LIN {X 0,Y 130.717,Z 907.03,A -85,B 0,C 180,E1 -25688.192,E2 -25688.192} C_VEL
LIN {X 0,Y 137.443,Z 899.876,A -85,B 0,C 180,E1 -25692.65,E2 -25692.65} C_VEL
LIN {X 0,Y 145.059,Z 891.056,A -85,B 0,C 180,E1 -25696.613,E2 -25696.613} C_VEL
LIN {X 0,Y 152.353,Z 881.374,A -85,B 0,C 180,E1 -25699.855,E2 -25699.855} C_VEL
LIN {X 0,Y 159.41,Z 870.654,A -85,B 0,C 180,E1 -25702.521,E2 -25702.521} C_VEL
LIN {X 0,Y 165.915,Z 859.265,A -85,B 0,C 180,E1 -25704.628,E2 -25704.628} C_VEL
LIN {X 0,Y 171.979,Z 846.674,A -85,B 0,C 180,E1 -25706.37,E2 -25706.37} C_VEL
LIN {X 0,Y 176.788,Z 834.475,A -85,B 0,C 180,E1 -25707.647,E2 -25707.647} C_VEL
LIN {X 0,Y 181.009,Z 821.027,A -85,B 0,C 180,E1 -25708.67,E2 -25708.67} C_VEL
LIN {X 0,Y 184.333,Z 806.496,A -85,B 0,C 180,E1 -25709.448,E2 -25709.448} C_VEL
LIN {X 0,Y 186.375,Z 792.089,A -85,B 0,C 180,E1 -25709.962,E2 -25709.962} C_VEL
LIN {X 0,Y 188.854,Z 764.424,A -85,B 0,C 180,E1 -25710.763,E2 -25710.763} C_VEL
LIN {X 0,Y 185.546,Z 755.043,A -85,B 0,C 180,E1 -25713.686,E2 -25713.686} C_VEL
LIN {X 0,Y 181.921,Z 745.913,A -85,B 0,C 180,E1 -25717.352,E2 -25717.352} C_VEL
LIN {X 0,Y 179.613,Z 740.879,A -85,B 0,C 180,E1 -25720.053,E2 -25720.053} C_VEL
LIN {X 0,Y 178.02,Z 738.111,A -85,B 0,C 180,E1 -25722.125,E2 -25722.125} C_VEL
LIN {X 0,Y 176.17,Z 734.921,A -85,B 0,C 180,E1 -25724.99,E2 -25724.99} C_VEL
LIN {X 0,Y 174.114,Z 731.175,A -85,B 0,C 180,E1 -25729.388,E2 -25729.388} C_VEL
LIN {X 0,Y 172.685,Z 729.526,A -85,B 0,C 180,E1 -25734.747,E2 -25734.747} C_VEL
LIN {X 0,Y 172.506,Z 728.977,A -85,B 0,C 180,E1 -25737.666,E2 -25737.666} C_VEL
LIN {X 0,Y 172.681,Z 729.24,A -85,B 0,C 180,E1 -25740.584,E2 -25740.584} C_VEL
LIN {X 0,Y 174.136,Z 731.139,A -85,B 0,C 180,E1 -25746.228,E2 -25746.228} C_VEL
LIN {X 0,Y 175.9,Z 734.558,A -85,B 0,C 180,E1 -25750.127,E2 -25750.127} C_VEL
LIN {X 0,Y 176.7,Z 735.811,A -85,B 0,C 180,E1 -25751.471,E2 -25751.471} C_VEL
LIN {X 0,Y 179.182,Z 740.077,A -85,B 0,C 180,E1 -25754.985,E2 -25754.985} C_VEL
LIN {X 0,Y 181.956,Z 744.921,A -85,B 0,C 180,E1 -25758.145,E2 -25758.145} C_VEL
LIN {X 0,Y 185.573,Z 751.685,A -85,B 0,C 180,E1 -25761.597,E2 -25761.597} C_VEL
LIN {X 0,Y 189.253,Z 759.361,A -85,B 0,C 180,E1 -25764.636,E2 -25764.636} C_VEL
LIN {X 0,Y 186.164,Z 792.33,A -85,B 0,C 180,E1 -25765.653,E2 -25765.653} C_VEL
LIN {X 0,Y 183.619,Z 806.633,A -85,B 0,C 180,E1 -25766.329,E2 -25766.329} C_VEL
LIN {X 0,Y 179.972,Z 820.763,A -85,B 0,C 180,E1 -25767.327,E2 -25767.327} C_VEL
LIN {X 0,Y 175.366,Z 833.914,A -85,B 0,C 180,E1 -25768.54,E2 -25768.54} C_VEL
LIN {X 0,Y 169.817,Z 846.919,A -85,B 0,C 180,E1 -25770.24,E2 -25770.24} C_VEL
LIN {X 0,Y 163.992,Z 858.202,A -85,B 0,C 180,E1 -25772.178,E2 -25772.178} C_VEL
LIN {X 0,Y 157.701,Z 868.563,A -85,B 0,C 180,E1 -25774.467,E2 -25774.467} C_VEL
LIN {X 0,Y 150.527,Z 878.834,A -85,B 0,C 180,E1 -25777.466,E2 -25777.466} C_VEL
LIN {X 0,Y 143.871,Z 887.3,A -85,B 0,C 180,E1 -25780.786,E2 -25780.786} C_VEL
LIN {X 0,Y 136.6,Z 895.355,A -85,B 0,C 180,E1 -25784.974,E2 -25784.974} C_VEL
LIN {X 0,Y 130.127,Z 901.821,A -85,B 0,C 180,E1 -25789.601,E2 -25789.601} C_VEL
LIN {X 0,Y 123.866,Z 907.527,A -85,B 0,C 180,E1 -25795.432,E2 -25795.432} C_VEL
LIN {X 0,Y 118.937,Z 911.65,A -85,B 0,C 180,E1 -25801.789,E2 -25801.789} C_VEL
LIN {X 0,Y 115.304,Z 914.323,A -85,B 0,C 180,E1 -25808.549,E2 -25808.549} C_VEL
LIN {X 0,Y 113.093,Z 915.631,A -85,B 0,C 180,E1 -25815.607,E2 -25815.607} C_VEL
LIN {X 0,Y 112.299,Z 915.605,A -85,B 0,C 180,E1 -25822.81,E2 -25822.81} C_VEL
LIN {X 0,Y 112.519,Z 914.265,A -85,B 0,C 180,E1 -25830,E2 -25830} C_VEL
LIN {X 0,Y 113.594,Z 911.605,A -85,B 0,C 180,E1 -25837.108,E2 -25837.108} C_VEL
LIN {X 0,Y 116.097,Z 907.532,A -85,B 0,C 180,E1 -25844.013,E2 -25844.013} C_VEL
LIN {X 0,Y 118.716,Z 903.661,A -85,B 0,C 180,E1 -25848.823,E2 -25848.823} C_VEL
LIN {X 0,Y 122.207,Z 898.494,A -85,B 0,C 180,E1 -25853.739,E2 -25853.739} C_VEL
LIN {X 0,Y 126.961,Z 891.34,A -85,B 0,C 180,E1 -25858.971,E2 -25858.971} C_VEL
LIN {X 0,Y 132.939,Z 882.461,A -85,B 0,C 180,E1 -25863.718,E2 -25863.718} C_VEL
LIN {X 0,Y 138.59,Z 873.147,A -85,B 0,C 180,E1 -25867.484,E2 -25867.484} C_VEL
LIN {X 0,Y 144.56,Z 861.8,A -85,B 0,C 180,E1 -25871.021,E2 -25871.021} C_VEL
LIN {X 0,Y 149.314,Z 851.519,A -85,B 0,C 180,E1 -25873.502,E2 -25873.502} C_VEL
LIN {X 0,Y 154.449,Z 838.934,A -85,B 0,C 180,E1 -25875.782,E2 -25875.782} C_VEL
LIN {X 0,Y 158.616,Z 826.703,A -85,B 0,C 180,E1 -25877.445,E2 -25877.445} C_VEL
LIN {X 0,Y 162.163,Z 813.199,A -85,B 0,C 180,E1 -25878.853,E2 -25878.853} C_VEL
LIN {X 0,Y 164.868,Z 799.207,A -85,B 0,C 180,E1 -25879.875,E2 -25879.875} C_VEL
LIN {X 0,Y 166.63,Z 784.548,A -85,B 0,C 180,E1 -25880.569,E2 -25880.569} C_VEL
LIN {X 0,Y 170.019,Z 743.584,A -85,B 0,C 180,E1 -25881.9,E2 -25881.9} C_VEL
LIN {X 0,Y 164.97,Z 733.193,A -85,B 0,C 180,E1 -25885.295,E2 -25885.295} C_VEL
LIN {X 0,Y 160.233,Z 724.666,A -85,B 0,C 180,E1 -25888.918,E2 -25888.918} C_VEL
LIN {X 0,Y 156.243,Z 718.002,A -85,B 0,C 180,E1 -25892.487,E2 -25892.487} C_VEL
LIN {X 0,Y 153.557,Z 713.992,A -85,B 0,C 180,E1 -25895.255,E2 -25895.255} C_VEL
LIN {X 0,Y 151.039,Z 710.195,A -85,B 0,C 180,E1 -25898.306,E2 -25898.306} C_VEL
LIN {X 0,Y 148.535,Z 706.642,A -85,B 0,C 180,E1 -25901.998,E2 -25901.998} C_VEL
LIN {X 0,Y 148.119,Z 705.866,A -85,B 0,C 180,E1 -25902.748,E2 -25902.748} C_VEL
LIN {X 0,Y 145.875,Z 703.314,A -85,B 0,C 180,E1 -25907.393,E2 -25907.393} C_VEL
LIN {X 0,Y 144.917,Z 700.704,A -85,B 0,C 180,E1 -25910.974,E2 -25910.974} C_VEL
LIN {X 0,Y 144.277,Z 700.177,A -85,B 0,C 180,E1 -25919.999,E2 -25919.999} C_VEL
LIN {X 0,Y 145.22,Z 701.037,A -85,B 0,C 180,E1 -25924.684,E2 -25924.684} C_VEL
LIN {X 0,Y 146.997,Z 704.735,A -85,B 0,C 180,E1 -25929.703,E2 -25929.703} C_VEL
LIN {X 0,Y 148.44,Z 706.253,A -85,B 0,C 180,E1 -25932.301,E2 -25932.301} C_VEL
LIN {X 0,Y 150.683,Z 709.743,A -85,B 0,C 180,E1 -25935.729,E2 -25935.729} C_VEL
LIN {X 0,Y 151.749,Z 711.247,A -85,B 0,C 180,E1 -25937.107,E2 -25937.107} C_VEL
LIN {X 0,Y 154.655,Z 715.613,A -85,B 0,C 180,E1 -25940.417,E2 -25940.417} C_VEL
LIN {X 0,Y 157.539,Z 720.16,A -85,B 0,C 180,E1 -25943.236,E2 -25943.236} C_VEL
LIN {X 0,Y 161.113,Z 726.258,A -85,B 0,C 180,E1 -25946.297,E2 -25946.297} C_VEL
LIN {X 0,Y 165.099,Z 735.997,A -85,B 0,C 180,E1 -25949.495,E2 -25949.495} C_VEL
LIN {X 0,Y 169.26,Z 747.65,A -85,B 0,C 180,E1 -25952.522,E2 -25952.522} C_VEL
LIN {X 0,Y 169.697,Z 749.178,A -85,B 0,C 180,E1 -25952.84,E2 -25952.84} C_VEL
LIN {X 0,Y 165.504,Z 798.715,A -85,B 0,C 180,E1 -25954.502,E2 -25954.502} C_VEL
LIN {X 0,Y 163.103,Z 813.487,A -85,B 0,C 180,E1 -25955.313,E2 -25955.313} C_VEL
LIN {X 0,Y 159.562,Z 828.086,A -85,B 0,C 180,E1 -25956.502,E2 -25956.502} C_VEL
LIN {X 0,Y 155.183,Z 841.89,A -85,B 0,C 180,E1 -25958.104,E2 -25958.104} C_VEL
LIN {X 0,Y 150.286,Z 854.269,A -85,B 0,C 180,E1 -25960.024,E2 -25960.024} C_VEL
LIN {X 0,Y 145.147,Z 865.623,A -85,B 0,C 180,E1 -25962.404,E2 -25962.404} C_VEL
LIN {X 0,Y 139.796,Z 876.072,A -85,B 0,C 180,E1 -25965.265,E2 -25965.265} C_VEL
LIN {X 0,Y 133.759,Z 886.452,A -85,B 0,C 180,E1 -25968.945,E2 -25968.945} C_VEL
LIN {X 0,Y 128.338,Z 895.029,A -85,B 0,C 180,E1 -25972.959,E2 -25972.959} C_VEL
LIN {X 0,Y 122.956,Z 903.223,A -85,B 0,C 180,E1 -25978.081,E2 -25978.081} C_VEL
LIN {X 0,Y 118.547,Z 909.826,A -85,B 0,C 180,E1 -25983.6,E2 -25983.6} C_VEL
LIN {X 0,Y 115.802,Z 914.416,A -85,B 0,C 180,E1 -25988.645,E2 -25988.645} C_VEL
LIN {X 0,Y 113.294,Z 919.053,A -85,B 0,C 180,E1 -25995.633,E2 -25995.633} C_VEL
LIN {X 0,Y 112.287,Z 922.199,A -85,B 0,C 180,E1 -26002.808,E2 -26002.808} C_VEL
LIN {X 0,Y 112.259,Z 923.245,A -85,B 0,C 180,E1 -26006.41,E2 -26006.41} C_VEL
LIN {X 0,Y 112.387,Z 923.943,A -85,B 0,C 180,E1 -26010,E2 -26010} C_VEL
LIN {X 0,Y 112.279,Z 924.28,A -85,B 0,C 180,E1 -26017.191,E2 -26017.191} C_VEL
LIN {X 0,Y 113.341,Z 923.284,A -85,B 0,C 180,E1 -26024.361,E2 -26024.361} C_VEL
LIN {X 0,Y 115.68,Z 921.177,A -85,B 0,C 180,E1 -26030.766,E2 -26030.766} C_VEL
LIN {X 0,Y 116.52,Z 919.969,A -85,B 0,C 180,E1 -26033.588,E2 -26033.588} C_VEL
LIN {X 0,Y 116.655,Z 917.511,A -85,B 0,C 180,E1 -26038.312,E2 -26038.312} C_VEL
LIN {X 0,Y 117.122,Z 915.124,A -85,B 0,C 180,E1 -26042.03,E2 -26042.03} C_VEL
LIN {X 0,Y 118.513,Z 913.086,A -85,B 0,C 180,E1 -26044.647,E2 -26044.647} C_VEL
LIN {X 0,Y 119.273,Z 912.338,A -85,B 0,C 180,E1 -26045.452,E2 -26045.452} C_VEL
LIN {X 0,Y 125.189,Z 906.907,A -85,B 0,C 180,E1 -26050.21,E2 -26050.21} C_VEL
LIN {X 0,Y 132.303,Z 899.79,A -85,B 0,C 180,E1 -26054.736,E2 -26054.736} C_VEL
LIN {X 0,Y 139.109,Z 892.367,A -85,B 0,C 180,E1 -26058.175,E2 -26058.175} C_VEL
LIN {X 0,Y 146.49,Z 883.189,A -85,B 0,C 180,E1 -26061.415,E2 -26061.415} C_VEL
LIN {X 0,Y 153.873,Z 872.716,A -85,B 0,C 180,E1 -26064.165,E2 -26064.165} C_VEL
LIN {X 0,Y 160.553,Z 861.846,A -85,B 0,C 180,E1 -26066.274,E2 -26066.274} C_VEL
LIN {X 0,Y 166.749,Z 849.962,A -85,B 0,C 180,E1 -26068.017,E2 -26068.017} C_VEL
LIN {X 0,Y 172.404,Z 836.826,A -85,B 0,C 180,E1 -26069.446,E2 -26069.446} C_VEL
